;FOLD PLACE 2
;FOLD PROPRIEDADES
Ponto_STR[Pallet_2,Prdt_32BarPacking,2].NumCaixas = 3
Ponto_STR[Pallet_2,Prdt_32BarPacking,2].PickOp = 2
Ponto_STR[Pallet_2,Prdt_32BarPacking,2].ConfGarraOp = 3
Ponto_STR[Pallet_2,Prdt_32BarPacking,2].FechaGarraOp = 0
Ponto_STR[Pallet_2,Prdt_32BarPacking,2].AbreGarraOp = 0
Ponto_STR[Pallet_2,Prdt_32BarPacking,2].SensoresCaixa = 12345
Ponto_STR[Pallet_2,Prdt_32BarPacking,2].TravaGarra = False
Ponto_STR[Pallet_2,Prdt_32BarPacking,2].SkipGoHome = False
Ponto_STR[Pallet_2,Prdt_32BarPacking,2].SkipSobeRelativo = False
Ponto_STR[Pallet_2,Prdt_32BarPacking,2].XApp1Place=P2_32BarPacking_2_App1
Ponto_STR[Pallet_2,Prdt_32BarPacking,2].XApp2Place=P2_32BarPacking_2_App2
Ponto_STR[Pallet_2,Prdt_32BarPacking,2].XPlace=P2_32BarPacking_2_Place
;ENDFOLD
;FOLD OffsetPlace
Ponto_STR[Pallet_2,Prdt_32BarPacking,2].OffsetPlace.X=0
Ponto_STR[Pallet_2,Prdt_32BarPacking,2].OffsetPlace.Y=0
Ponto_STR[Pallet_2,Prdt_32BarPacking,2].OffsetPlace.Z=0
Ponto_STR[Pallet_2,Prdt_32BarPacking,2].OffsetPlace.A=0
Ponto_STR[Pallet_2,Prdt_32BarPacking,2].OffsetPlace.B=0
Ponto_STR[Pallet_2,Prdt_32BarPacking,2].OffsetPlace.C=0
;ENDFOLD
;ENDFOLD

;FOLD PLACE 3
;FOLD PROPRIEDADES
Ponto_STR[Pallet_2,Prdt_32BarPacking,3].NumCaixas = 3
Ponto_STR[Pallet_2,Prdt_32BarPacking,3].PickOp = 2
Ponto_STR[Pallet_2,Prdt_32BarPacking,3].ConfGarraOp = 3
Ponto_STR[Pallet_2,Prdt_32BarPacking,3].FechaGarraOp = 0
Ponto_STR[Pallet_2,Prdt_32BarPacking,3].AbreGarraOp = 0
Ponto_STR[Pallet_2,Prdt_32BarPacking,3].SensoresCaixa = 12345
Ponto_STR[Pallet_2,Prdt_32BarPacking,3].TravaGarra = False
Ponto_STR[Pallet_2,Prdt_32BarPacking,3].SkipGoHome = False
Ponto_STR[Pallet_2,Prdt_32BarPacking,3].SkipSobeRelativo = False
Ponto_STR[Pallet_2,Prdt_32BarPacking,3].XApp1Place=P2_32BarPacking_3_App1
Ponto_STR[Pallet_2,Prdt_32BarPacking,3].XApp2Place=P2_32BarPacking_3_App2
Ponto_STR[Pallet_2,Prdt_32BarPacking,3].XPlace=P2_32BarPacking_3_Place
;ENDFOLD
;FOLD OffsetPlace
Ponto_STR[Pallet_2,Prdt_32BarPacking,3].OffsetPlace.X=0
Ponto_STR[Pallet_2,Prdt_32BarPacking,3].OffsetPlace.Y=0
Ponto_STR[Pallet_2,Prdt_32BarPacking,3].OffsetPlace.Z=0
Ponto_STR[Pallet_2,Prdt_32BarPacking,3].OffsetPlace.A=0
Ponto_STR[Pallet_2,Prdt_32BarPacking,3].OffsetPlace.B=0
Ponto_STR[Pallet_2,Prdt_32BarPacking,3].OffsetPlace.C=0
;ENDFOLD
;ENDFOLD

;ENDFOLD
;ENDFOLD

;FOLD Pallet 2 - Produto 33BarPacking
;FOLD LAYER 1: PLACE 1 ate 2
;FOLD PLACE 1
;FOLD PROPRIEDADES
Ponto_STR[Pallet_2,Prdt_33BarPacking,1].NumCaixas = 3
Ponto_STR[Pallet_2,Prdt_33BarPacking,1].PickOp = 2
Ponto_STR[Pallet_2,Prdt_33BarPacking,1].ConfGarraOp = 2
Ponto_STR[Pallet_2,Prdt_33BarPacking,1].FechaGarraOp = 0
Ponto_STR[Pallet_2,Prdt_33BarPacking,1].AbreGarraOp = 0
Ponto_STR[Pallet_2,Prdt_33BarPacking,1].SensoresCaixa = 12345
Ponto_STR[Pallet_2,Prdt_33BarPacking,1].TravaGarra = False
Ponto_STR[Pallet_2,Prdt_33BarPacking,1].SkipGoHome = False
Ponto_STR[Pallet_2,Prdt_33BarPacking,1].SkipSobeRelativo = False
Ponto_STR[Pallet_2,Prdt_33BarPacking,1].XApp1Place=P2_33BarPacking_1_App1
Ponto_STR[Pallet_2,Prdt_33BarPacking,1].XApp2Place=P2_33BarPacking_1_App2
Ponto_STR[Pallet_2,Prdt_33BarPacking,1].XPlace=P2_33BarPacking_1_Place
;ENDFOLD
;FOLD OffsetPlace
Ponto_STR[Pallet_2,Prdt_33BarPacking,1].OffsetPlace.X=0
Ponto_STR[Pallet_2,Prdt_33BarPacking,1].OffsetPlace.Y=0
Ponto_STR[Pallet_2,Prdt_33BarPacking,1].OffsetPlace.Z=0
Ponto_STR[Pallet_2,Prdt_33BarPacking,1].OffsetPlace.A=0
Ponto_STR[Pallet_2,Prdt_33BarPacking,1].OffsetPlace.B=0
Ponto_STR[Pallet_2,Prdt_33BarPacking,1].OffsetPlace.C=0
;ENDFOLD
;ENDFOLD

;FOLD PLACE 2
;FOLD PROPRIEDADES
Ponto_STR[Pallet_2,Prdt_33BarPacking,2].NumCaixas = 3
Ponto_STR[Pallet_2,Prdt_33BarPacking,2].PickOp = 2
Ponto_STR[Pallet_2,Prdt_33BarPacking,2].ConfGarraOp = 2
Ponto_STR[Pallet_2,Prdt_33BarPacking,2].FechaGarraOp = 0
Ponto_STR[Pallet_2,Prdt_33BarPacking,2].AbreGarraOp = 0
Ponto_STR[Pallet_2,Prdt_33BarPacking,2].SensoresCaixa = 12345
Ponto_STR[Pallet_2,Prdt_33BarPacking,2].TravaGarra = False
Ponto_STR[Pallet_2,Prdt_33BarPacking,2].SkipGoHome = False
Ponto_STR[Pallet_2,Prdt_33BarPacking,2].SkipSobeRelativo = False
Ponto_STR[Pallet_2,Prdt_33BarPacking,2].XApp1Place=P2_33BarPacking_2_App1
Ponto_STR[Pallet_2,Prdt_33BarPacking,2].XApp2Place=P2_33BarPacking_2_App2
Ponto_STR[Pallet_2,Prdt_33BarPacking,2].XPlace=P2_33BarPacking_2_Place
;ENDFOLD
;FOLD OffsetPlace
Ponto_STR[Pallet_2,Prdt_33BarPacking,2].OffsetPlace.X=0
Ponto_STR[Pallet_2,Prdt_33BarPacking,2].OffsetPlace.Y=0
Ponto_STR[Pallet_2,Prdt_33BarPacking,2].OffsetPlace.Z=0
Ponto_STR[Pallet_2,Prdt_33BarPacking,2].OffsetPlace.A=0
Ponto_STR[Pallet_2,Prdt_33BarPacking,2].OffsetPlace.B=0
Ponto_STR[Pallet_2,Prdt_33BarPacking,2].OffsetPlace.C=0
;ENDFOLD
;ENDFOLD

;ENDFOLD
;ENDFOLD

;FOLD Pallet 2 - Produto 34BarPacking
;FOLD LAYER 1: PLACE 1 ate 2
;FOLD PLACE 1
;FOLD PROPRIEDADES
Ponto_STR[Pallet_2,Prdt_34BarPacking,1].NumCaixas = 1
Ponto_STR[Pallet_2,Prdt_34BarPacking,1].PickOp = 3
Ponto_STR[Pallet_2,Prdt_34BarPacking,1].ConfGarraOp = 3
Ponto_STR[Pallet_2,Prdt_34BarPacking,1].FechaGarraOp = 0
Ponto_STR[Pallet_2,Prdt_34BarPacking,1].AbreGarraOp = 0
Ponto_STR[Pallet_2,Prdt_34BarPacking,1].SensoresCaixa = 123
Ponto_STR[Pallet_2,Prdt_34BarPacking,1].TravaGarra = False
Ponto_STR[Pallet_2,Prdt_34BarPacking,1].SkipGoHome = False
Ponto_STR[Pallet_2,Prdt_34BarPacking,1].SkipSobeRelativo = False
Ponto_STR[Pallet_2,Prdt_34BarPacking,1].XApp1Place=P2_34BarPacking_1_App1
Ponto_STR[Pallet_2,Prdt_34BarPacking,1].XApp2Place=P2_34BarPacking_1_App2
Ponto_STR[Pallet_2,Prdt_34BarPacking,1].XPlace=P2_34BarPacking_1_Place
;ENDFOLD
;FOLD OffsetPlace
Ponto_STR[Pallet_2,Prdt_34BarPacking,1].OffsetPlace.X=0
Ponto_STR[Pallet_2,Prdt_34BarPacking,1].OffsetPlace.Y=0
Ponto_STR[Pallet_2,Prdt_34BarPacking,1].OffsetPlace.Z=0
Ponto_STR[Pallet_2,Prdt_34BarPacking,1].OffsetPlace.A=0
Ponto_STR[Pallet_2,Prdt_34BarPacking,1].OffsetPlace.B=0
Ponto_STR[Pallet_2,Prdt_34BarPacking,1].OffsetPlace.C=0
;ENDFOLD
;ENDFOLD

;FOLD PLACE 2
;FOLD PROPRIEDADES
Ponto_STR[Pallet_2,Prdt_34BarPacking,2].NumCaixas = 1
Ponto_STR[Pallet_2,Prdt_34BarPacking,2].PickOp = 3
Ponto_STR[Pallet_2,Prdt_34BarPacking,2].ConfGarraOp = 3
Ponto_STR[Pallet_2,Prdt_34BarPacking,2].FechaGarraOp = 0
Ponto_STR[Pallet_2,Prdt_34BarPacking,2].AbreGarraOp = 0
Ponto_STR[Pallet_2,Prdt_34BarPacking,2].SensoresCaixa = 123
Ponto_STR[Pallet_2,Prdt_34BarPacking,2].TravaGarra = False
Ponto_STR[Pallet_2,Prdt_34BarPacking,2].SkipGoHome = False
Ponto_STR[Pallet_2,Prdt_34BarPacking,2].SkipSobeRelativo = False
Ponto_STR[Pallet_2,Prdt_34BarPacking,2].XApp1Place=P2_34BarPacking_2_App1
Ponto_STR[Pallet_2,Prdt_34BarPacking,2].XApp2Place=P2_34BarPacking_2_App2
Ponto_STR[Pallet_2,Prdt_34BarPacking,2].XPlace=P2_34BarPacking_2_Place
;ENDFOLD
;FOLD OffsetPlace
Ponto_STR[Pallet_2,Prdt_34BarPacking,2].OffsetPlace.X=0
Ponto_STR[Pallet_2,Prdt_34BarPacking,2].OffsetPlace.Y=0
Ponto_STR[Pallet_2,Prdt_34BarPacking,2].OffsetPlace.Z=0
Ponto_STR[Pallet_2,Prdt_34BarPacking,2].OffsetPlace.A=0
Ponto_STR[Pallet_2,Prdt_34BarPacking,2].OffsetPlace.B=0
Ponto_STR[Pallet_2,Prdt_34BarPacking,2].OffsetPlace.C=0
;ENDFOLD
;ENDFOLD

;ENDFOLD
;ENDFOLD

;FOLD Pallet 2 - Produto 9Aero
;FOLD LAYER 1: PLACE 1 ate 2
;FOLD PLACE 1
;FOLD PROPRIEDADES
Ponto_STR[Pallet_2,Prdt_9Aero,1].NumCaixas = 4
Ponto_STR[Pallet_2,Prdt_9Aero,1].PickOp = 3
Ponto_STR[Pallet_2,Prdt_9Aero,1].ConfGarraOp = 3
Ponto_STR[Pallet_2,Prdt_9Aero,1].FechaGarraOp = 0
Ponto_STR[Pallet_2,Prdt_9Aero,1].AbreGarraOp = 0
Ponto_STR[Pallet_2,Prdt_9Aero,1].SensoresCaixa = 123456
Ponto_STR[Pallet_2,Prdt_9Aero,1].TravaGarra = False
Ponto_STR[Pallet_2,Prdt_9Aero,1].SkipGoHome = False
Ponto_STR[Pallet_2,Prdt_9Aero,1].SkipSobeRelativo = False
Ponto_STR[Pallet_2,Prdt_9Aero,1].XApp1Place=P2_9Aero_1_App1
Ponto_STR[Pallet_2,Prdt_9Aero,1].XApp2Place=P2_9Aero_1_App2
Ponto_STR[Pallet_2,Prdt_9Aero,1].XPlace=P2_9Aero_1_Place
;ENDFOLD
;FOLD OffsetPlace
Ponto_STR[Pallet_2,Prdt_9Aero,1].OffsetPlace.X=0
Ponto_STR[Pallet_2,Prdt_9Aero,1].OffsetPlace.Y=0
Ponto_STR[Pallet_2,Prdt_9Aero,1].OffsetPlace.Z=0
Ponto_STR[Pallet_2,Prdt_9Aero,1].OffsetPlace.A=0
Ponto_STR[Pallet_2,Prdt_9Aero,1].OffsetPlace.B=0
Ponto_STR[Pallet_2,Prdt_9Aero,1].OffsetPlace.C=0
;ENDFOLD
;ENDFOLD

;FOLD PLACE 2
;FOLD PROPRIEDADES
Ponto_STR[Pallet_2,Prdt_9Aero,2].NumCaixas = 4
Ponto_STR[Pallet_2,Prdt_9Aero,2].PickOp = 3
Ponto_STR[Pallet_2,Prdt_9Aero,2].ConfGarraOp = 3
Ponto_STR[Pallet_2,Prdt_9Aero,2].FechaGarraOp = 0
Ponto_STR[Pallet_2,Prdt_9Aero,2].AbreGarraOp = 0
Ponto_STR[Pallet_2,Prdt_9Aero,2].SensoresCaixa = 123456
Ponto_STR[Pallet_2,Prdt_9Aero,2].TravaGarra = False
Ponto_STR[Pallet_2,Prdt_9Aero,2].SkipGoHome = False
Ponto_STR[Pallet_2,Prdt_9Aero,2].SkipSobeRelativo = False
Ponto_STR[Pallet_2,Prdt_9Aero,2].XApp1Place=P2_9Aero_2_App1
Ponto_STR[Pallet_2,Prdt_9Aero,2].XApp2Place=P2_9Aero_2_App2
Ponto_STR[Pallet_2,Prdt_9Aero,2].XPlace=P2_9Aero_2_Place
;ENDFOLD
;FOLD OffsetPlace
Ponto_STR[Pallet_2,Prdt_9Aero,2].OffsetPlace.X=0
Ponto_STR[Pallet_2,Prdt_9Aero,2].OffsetPlace.Y=0
Ponto_STR[Pallet_2,Prdt_9Aero,2].OffsetPlace.Z=0
Ponto_STR[Pallet_2,Prdt_9Aero,2].OffsetPlace.A=0
Ponto_STR[Pallet_2,Prdt_9Aero,2].OffsetPlace.B=0
Ponto_STR[Pallet_2,Prdt_9Aero,2].OffsetPlace.C=0
;ENDFOLD
;ENDFOLD

;ENDFOLD
;ENDFOLD

;FOLD Pallet 2 - Produto 23Smarties
;FOLD LAYER 1: PLACE 1 ate 4
;FOLD PLACE 1
;FOLD PROPRIEDADES
Ponto_STR[Pallet_2,Prdt_23Smarties,1].NumCaixas = 2
Ponto_STR[Pallet_2,Prdt_23Smarties,1].PickOp = 4
Ponto_STR[Pallet_2,Prdt_23Smarties,1].ConfGarraOp = 4
Ponto_STR[Pallet_2,Prdt_23Smarties,1].FechaGarraOp = 0
Ponto_STR[Pallet_2,Prdt_23Smarties,1].AbreGarraOp = 0
Ponto_STR[Pallet_2,Prdt_23Smarties,1].SensoresCaixa = 456
Ponto_STR[Pallet_2,Prdt_23Smarties,1].TravaGarra = False
Ponto_STR[Pallet_2,Prdt_23Smarties,1].SkipGoHome = False
Ponto_STR[Pallet_2,Prdt_23Smarties,1].SkipSobeRelativo = False
Ponto_STR[Pallet_2,Prdt_23Smarties,1].XApp1Place=P2_23Smarties_1_App1
Ponto_STR[Pallet_2,Prdt_23Smarties,1].XApp2Place=P2_23Smarties_1_App2
Ponto_STR[Pallet_2,Prdt_23Smarties,1].XPlace=P2_23Smarties_1_Place
;ENDFOLD
;FOLD OffsetPlace
Ponto_STR[Pallet_2,Prdt_23Smarties,1].OffsetPlace.X=0
Ponto_STR[Pallet_2,Prdt_23Smarties,1].OffsetPlace.Y=0
Ponto_STR[Pallet_2,Prdt_23Smarties,1].OffsetPlace.Z=0
Ponto_STR[Pallet_2,Prdt_23Smarties,1].OffsetPlace.A=0
Ponto_STR[Pallet_2,Prdt_23Smarties,1].OffsetPlace.B=0
Ponto_STR[Pallet_2,Prdt_23Smarties,1].OffsetPlace.C=0
;ENDFOLD
;ENDFOLD

;FOLD PLACE 2
;FOLD PROPRIEDADES
Ponto_STR[Pallet_2,Prdt_23Smarties,2].NumCaixas = 3
Ponto_STR[Pallet_2,Prdt_23Smarties,2].PickOp = 4
Ponto_STR[Pallet_2,Prdt_23Smarties,2].ConfGarraOp = 4
Ponto_STR[Pallet_2,Prdt_23Smarties,2].FechaGarraOp = 0
Ponto_STR[Pallet_2,Prdt_23Smarties,2].AbreGarraOp = 0
Ponto_STR[Pallet_2,Prdt_23Smarties,2].SensoresCaixa = 3456
Ponto_STR[Pallet_2,Prdt_23Smarties,2].TravaGarra = False
Ponto_STR[Pallet_2,Prdt_23Smarties,2].SkipGoHome = False
Ponto_STR[Pallet_2,Prdt_23Smarties,2].SkipSobeRelativo = False
Ponto_STR[Pallet_2,Prdt_23Smarties,2].XApp1Place=P2_23Smarties_2_App1
Ponto_STR[Pallet_2,Prdt_23Smarties,2].XApp2Place=P2_23Smarties_2_App2
Ponto_STR[Pallet_2,Prdt_23Smarties,2].XPlace=P2_23Smarties_2_Place
;ENDFOLD
;FOLD OffsetPlace
Ponto_STR[Pallet_2,Prdt_23Smarties,2].OffsetPlace.X=0
Ponto_STR[Pallet_2,Prdt_23Smarties,2].OffsetPlace.Y=0
Ponto_STR[Pallet_2,Prdt_23Smarties,2].OffsetPlace.Z=0
Ponto_STR[Pallet_2,Prdt_23Smarties,2].OffsetPlace.A=0
Ponto_STR[Pallet_2,Prdt_23Smarties,2].OffsetPlace.B=0
Ponto_STR[Pallet_2,Prdt_23Smarties,2].OffsetPlace.C=0
;ENDFOLD
;ENDFOLD

;FOLD PLACE 3
;FOLD PROPRIEDADES
Ponto_STR[Pallet_2,Prdt_23Smarties,3].NumCaixas = 2
Ponto_STR[Pallet_2,Prdt_23Smarties,3].PickOp = 4
Ponto_STR[Pallet_2,Prdt_23Smarties,3].ConfGarraOp = 4
Ponto_STR[Pallet_2,Prdt_23Smarties,3].FechaGarraOp = 0
Ponto_STR[Pallet_2,Prdt_23Smarties,3].AbreGarraOp = 0
Ponto_STR[Pallet_2,Prdt_23Smarties,3].SensoresCaixa = 456
Ponto_STR[Pallet_2,Prdt_23Smarties,3].TravaGarra = False
Ponto_STR[Pallet_2,Prdt_23Smarties,3].SkipGoHome = False
Ponto_STR[Pallet_2,Prdt_23Smarties,3].SkipSobeRelativo = False
Ponto_STR[Pallet_2,Prdt_23Smarties,3].XApp1Place=P2_23Smarties_3_App1
Ponto_STR[Pallet_2,Prdt_23Smarties,3].XApp2Place=P2_23Smarties_3_App2
Ponto_STR[Pallet_2,Prdt_23Smarties,3].XPlace=P2_23Smarties_3_Place
;ENDFOLD
;FOLD OffsetPlace
Ponto_STR[Pallet_2,Prdt_23Smarties,3].OffsetPlace.X=0
Ponto_STR[Pallet_2,Prdt_23Smarties,3].OffsetPlace.Y=0
Ponto_STR[Pallet_2,Prdt_23Smarties,3].OffsetPlace.Z=0
Ponto_STR[Pallet_2,Prdt_23Smarties,3].OffsetPlace.A=0
Ponto_STR[Pallet_2,Prdt_23Smarties,3].OffsetPlace.B=0
Ponto_STR[Pallet_2,Prdt_23Smarties,3].OffsetPlace.C=0
;ENDFOLD
;ENDFOLD

;FOLD PLACE 4
;FOLD PROPRIEDADES
Ponto_STR[Pallet_2,Prdt_23Smarties,4].NumCaixas = 3
Ponto_STR[Pallet_2,Prdt_23Smarties,4].PickOp = 4
Ponto_STR[Pallet_2,Prdt_23Smarties,4].ConfGarraOp = 4
Ponto_STR[Pallet_2,Prdt_23Smarties,4].FechaGarraOp = 0
Ponto_STR[Pallet_2,Prdt_23Smarties,4].AbreGarraOp = 0
Ponto_STR[Pallet_2,Prdt_23Smarties,4].SensoresCaixa = 3456
Ponto_STR[Pallet_2,Prdt_23Smarties,4].TravaGarra = False
Ponto_STR[Pallet_2,Prdt_23Smarties,4].SkipGoHome = False
Ponto_STR[Pallet_2,Prdt_23Smarties,4].SkipSobeRelativo = False
Ponto_STR[Pallet_2,Prdt_23Smarties,4].XApp1Place=P2_23Smarties_4_App1
Ponto_STR[Pallet_2,Prdt_23Smarties,4].XApp2Place=P2_23Smarties_4_App2
Ponto_STR[Pallet_2,Prdt_23Smarties,4].XPlace=P2_23Smarties_4_Place
;ENDFOLD
;FOLD OffsetPlace
Ponto_STR[Pallet_2,Prdt_23Smarties,4].OffsetPlace.X=0
Ponto_STR[Pallet_2,Prdt_23Smarties,4].OffsetPlace.Y=0
Ponto_STR[Pallet_2,Prdt_23Smarties,4].OffsetPlace.Z=0
Ponto_STR[Pallet_2,Prdt_23Smarties,4].OffsetPlace.A=0
Ponto_STR[Pallet_2,Prdt_23Smarties,4].OffsetPlace.B=0
Ponto_STR[Pallet_2,Prdt_23Smarties,4].OffsetPlace.C=0
;ENDFOLD
;ENDFOLD

;ENDFOLD
;FOLD LAYER 2: PLACE 5 ate 8
;FOLD PLACE 5
;FOLD PROPRIEDADES
Ponto_STR[Pallet_2,Prdt_23Smarties,5].NumCaixas = 2
Ponto_STR[Pallet_2,Prdt_23Smarties,5].PickOp = 5
Ponto_STR[Pallet_2,Prdt_23Smarties,5].ConfGarraOp = 4
Ponto_STR[Pallet_2,Prdt_23Smarties,5].FechaGarraOp = 0
Ponto_STR[Pallet_2,Prdt_23Smarties,5].AbreGarraOp = 0
Ponto_STR[Pallet_2,Prdt_23Smarties,5].SensoresCaixa = 123
Ponto_STR[Pallet_2,Prdt_23Smarties,5].TravaGarra = False
Ponto_STR[Pallet_2,Prdt_23Smarties,5].SkipGoHome = False
Ponto_STR[Pallet_2,Prdt_23Smarties,5].SkipSobeRelativo = False
Ponto_STR[Pallet_2,Prdt_23Smarties,5].XApp1Place=P2_23Smarties_5_App1
Ponto_STR[Pallet_2,Prdt_23Smarties,5].XApp2Place=P2_23Smarties_5_App2
Ponto_STR[Pallet_2,Prdt_23Smarties,5].XPlace=P2_23Smarties_5_Place
;ENDFOLD
;FOLD OffsetPlace
Ponto_STR[Pallet_2,Prdt_23Smarties,5].OffsetPlace.X=0
Ponto_STR[Pallet_2,Prdt_23Smarties,5].OffsetPlace.Y=0
Ponto_STR[Pallet_2,Prdt_23Smarties,5].OffsetPlace.Z=0
Ponto_STR[Pallet_2,Prdt_23Smarties,5].OffsetPlace.A=0
Ponto_STR[Pallet_2,Prdt_23Smarties,5].OffsetPlace.B=0
Ponto_STR[Pallet_2,Prdt_23Smarties,5].OffsetPlace.C=0
;ENDFOLD
;ENDFOLD

;FOLD PLACE 6
;FOLD PROPRIEDADES
Ponto_STR[Pallet_2,Prdt_23Smarties,6].NumCaixas = 3
Ponto_STR[Pallet_2,Prdt_23Smarties,6].PickOp = 5
Ponto_STR[Pallet_2,Prdt_23Smarties,6].ConfGarraOp = 4
Ponto_STR[Pallet_2,Prdt_23Smarties,6].FechaGarraOp = 0
Ponto_STR[Pallet_2,Prdt_23Smarties,6].AbreGarraOp = 0
Ponto_STR[Pallet_2,Prdt_23Smarties,6].SensoresCaixa = 1234
Ponto_STR[Pallet_2,Prdt_23Smarties,6].TravaGarra = False
Ponto_STR[Pallet_2,Prdt_23Smarties,6].SkipGoHome = False
Ponto_STR[Pallet_2,Prdt_23Smarties,6].SkipSobeRelativo = False
Ponto_STR[Pallet_2,Prdt_23Smarties,6].XApp1Place=P2_23Smarties_6_App1
Ponto_STR[Pallet_2,Prdt_23Smarties,6].XApp2Place=P2_23Smarties_6_App2
Ponto_STR[Pallet_2,Prdt_23Smarties,6].XPlace=P2_23Smarties_6_Place
;ENDFOLD
;FOLD OffsetPlace
Ponto_STR[Pallet_2,Prdt_23Smarties,6].OffsetPlace.X=0
Ponto_STR[Pallet_2,Prdt_23Smarties,6].OffsetPlace.Y=0
Ponto_STR[Pallet_2,Prdt_23Smarties,6].OffsetPlace.Z=0
Ponto_STR[Pallet_2,Prdt_23Smarties,6].OffsetPlace.A=0
Ponto_STR[Pallet_2,Prdt_23Smarties,6].OffsetPlace.B=0
Ponto_STR[Pallet_2,Prdt_23Smarties,6].OffsetPlace.C=0
;ENDFOLD
;ENDFOLD

;FOLD PLACE 7
;FOLD PROPRIEDADES
Ponto_STR[Pallet_2,Prdt_23Smarties,7].NumCaixas = 2
Ponto_STR[Pallet_2,Prdt_23Smarties,7].PickOp = 5
Ponto_STR[Pallet_2,Prdt_23Smarties,7].ConfGarraOp = 4
Ponto_STR[Pallet_2,Prdt_23Smarties,7].FechaGarraOp = 0
Ponto_STR[Pallet_2,Prdt_23Smarties,7].AbreGarraOp = 0
Ponto_STR[Pallet_2,Prdt_23Smarties,7].SensoresCaixa = 123
Ponto_STR[Pallet_2,Prdt_23Smarties,7].TravaGarra = False
Ponto_STR[Pallet_2,Prdt_23Smarties,7].SkipGoHome = False
Ponto_STR[Pallet_2,Prdt_23Smarties,7].SkipSobeRelativo = False
Ponto_STR[Pallet_2,Prdt_23Smarties,7].XApp1Place=P2_23Smarties_7_App1
Ponto_STR[Pallet_2,Prdt_23Smarties,7].XApp2Place=P2_23Smarties_7_App2
Ponto_STR[Pallet_2,Prdt_23Smarties,7].XPlace=P2_23Smarties_7_Place
;ENDFOLD
;FOLD OffsetPlace
Ponto_STR[Pallet_2,Prdt_23Smarties,7].OffsetPlace.X=0
Ponto_STR[Pallet_2,Prdt_23Smarties,7].OffsetPlace.Y=0
Ponto_STR[Pallet_2,Prdt_23Smarties,7].OffsetPlace.Z=0
Ponto_STR[Pallet_2,Prdt_23Smarties,7].OffsetPlace.A=0
Ponto_STR[Pallet_2,Prdt_23Smarties,7].OffsetPlace.B=0
Ponto_STR[Pallet_2,Prdt_23Smarties,7].OffsetPlace.C=0
;ENDFOLD
;ENDFOLD

;FOLD PLACE 8
;FOLD PROPRIEDADES
Ponto_STR[Pallet_2,Prdt_23Smarties,8].NumCaixas = 3
Ponto_STR[Pallet_2,Prdt_23Smarties,8].PickOp = 5
Ponto_STR[Pallet_2,Prdt_23Smarties,8].ConfGarraOp = 4
Ponto_STR[Pallet_2,Prdt_23Smarties,8].FechaGarraOp = 0
Ponto_STR[Pallet_2,Prdt_23Smarties,8].AbreGarraOp = 0
Ponto_STR[Pallet_2,Prdt_23Smarties,8].SensoresCaixa = 1234
Ponto_STR[Pallet_2,Prdt_23Smarties,8].TravaGarra = False
Ponto_STR[Pallet_2,Prdt_23Smarties,8].SkipGoHome = False
Ponto_STR[Pallet_2,Prdt_23Smarties,8].SkipSobeRelativo = False
Ponto_STR[Pallet_2,Prdt_23Smarties,8].XApp1Place=P2_23Smarties_8_App1
Ponto_STR[Pallet_2,Prdt_23Smarties,8].XApp2Place=P2_23Smarties_8_App2
Ponto_STR[Pallet_2,Prdt_23Smarties,8].XPlace=P2_23Smarties_8_Place
;ENDFOLD
;FOLD OffsetPlace
Ponto_STR[Pallet_2,Prdt_23Smarties,8].OffsetPlace.X=0
Ponto_STR[Pallet_2,Prdt_23Smarties,8].OffsetPlace.Y=0
Ponto_STR[Pallet_2,Prdt_23Smarties,8].OffsetPlace.Z=0
Ponto_STR[Pallet_2,Prdt_23Smarties,8].OffsetPlace.A=0
Ponto_STR[Pallet_2,Prdt_23Smarties,8].OffsetPlace.B=0
Ponto_STR[Pallet_2,Prdt_23Smarties,8].OffsetPlace.C=0
;ENDFOLD
;ENDFOLD

;ENDFOLD
;ENDFOLD

;FOLD Pallet 2 - Produto 10CoffeCrisp
;FOLD LAYER 1: PLACE 1 ate 4
;FOLD PLACE 1
;FOLD PROPRIEDADES
Ponto_STR[Pallet_2,Prdt_10CoffeCrisp,1].NumCaixas = 1
Ponto_STR[Pallet_2,Prdt_10CoffeCrisp,1].PickOp = 6
Ponto_STR[Pallet_2,Prdt_10CoffeCrisp,1].ConfGarraOp = 0
Ponto_STR[Pallet_2,Prdt_10CoffeCrisp,1].FechaGarraOp = 0
Ponto_STR[Pallet_2,Prdt_10CoffeCrisp,1].AbreGarraOp = 0
Ponto_STR[Pallet_2,Prdt_10CoffeCrisp,1].SensoresCaixa = 56
Ponto_STR[Pallet_2,Prdt_10CoffeCrisp,1].TravaGarra = False
Ponto_STR[Pallet_2,Prdt_10CoffeCrisp,1].SkipGoHome = False
Ponto_STR[Pallet_2,Prdt_10CoffeCrisp,1].SkipSobeRelativo = False
Ponto_STR[Pallet_2,Prdt_10CoffeCrisp,1].XApp1Place=P2_10CoffeCrisp_1_App1
Ponto_STR[Pallet_2,Prdt_10CoffeCrisp,1].XApp2Place=P2_10CoffeCrisp_1_App2
Ponto_STR[Pallet_2,Prdt_10CoffeCrisp,1].XPlace=P2_10CoffeCrisp_1_Place
;ENDFOLD
;FOLD OffsetPlace
Ponto_STR[Pallet_2,Prdt_10CoffeCrisp,1].OffsetPlace.X=0
Ponto_STR[Pallet_2,Prdt_10CoffeCrisp,1].OffsetPlace.Y=0
Ponto_STR[Pallet_2,Prdt_10CoffeCrisp,1].OffsetPlace.Z=0
Ponto_STR[Pallet_2,Prdt_10CoffeCrisp,1].OffsetPlace.A=0
Ponto_STR[Pallet_2,Prdt_10CoffeCrisp,1].OffsetPlace.B=0
Ponto_STR[Pallet_2,Prdt_10CoffeCrisp,1].OffsetPlace.C=0
;ENDFOLD
;ENDFOLD

;FOLD PLACE 2
;FOLD PROPRIEDADES
Ponto_STR[Pallet_2,Prdt_10CoffeCrisp,2].NumCaixas = 1
Ponto_STR[Pallet_2,Prdt_10CoffeCrisp,2].PickOp = 6
Ponto_STR[Pallet_2,Prdt_10CoffeCrisp,2].ConfGarraOp = 0
Ponto_STR[Pallet_2,Prdt_10CoffeCrisp,2].FechaGarraOp = 0
Ponto_STR[Pallet_2,Prdt_10CoffeCrisp,2].AbreGarraOp = 0
Ponto_STR[Pallet_2,Prdt_10CoffeCrisp,2].SensoresCaixa = 56
Ponto_STR[Pallet_2,Prdt_10CoffeCrisp,2].TravaGarra = False
Ponto_STR[Pallet_2,Prdt_10CoffeCrisp,2].SkipGoHome = False
Ponto_STR[Pallet_2,Prdt_10CoffeCrisp,2].SkipSobeRelativo = False
Ponto_STR[Pallet_2,Prdt_10CoffeCrisp,2].XApp1Place=P2_10CoffeCrisp_2_App1
Ponto_STR[Pallet_2,Prdt_10CoffeCrisp,2].XApp2Place=P2_10CoffeCrisp_2_App2
Ponto_STR[Pallet_2,Prdt_10CoffeCrisp,2].XPlace=P2_10CoffeCrisp_2_Place
;ENDFOLD
;FOLD OffsetPlace
Ponto_STR[Pallet_2,Prdt_10CoffeCrisp,2].OffsetPlace.X=0
Ponto_STR[Pallet_2,Prdt_10CoffeCrisp,2].OffsetPlace.Y=0
Ponto_STR[Pallet_2,Prdt_10CoffeCrisp,2].OffsetPlace.Z=0
Ponto_STR[Pallet_2,Prdt_10CoffeCrisp,2].OffsetPlace.A=0
Ponto_STR[Pallet_2,Prdt_10CoffeCrisp,2].OffsetPlace.B=0
Ponto_STR[Pallet_2,Prdt_10CoffeCrisp,2].OffsetPlace.C=0
;ENDFOLD
;ENDFOLD

;FOLD PLACE 3
;FOLD PROPRIEDADES
Ponto_STR[Pallet_2,Prdt_10CoffeCrisp,3].NumCaixas = 3
Ponto_STR[Pallet_2,Prdt_10CoffeCrisp,3].PickOp = 1
Ponto_STR[Pallet_2,Prdt_10CoffeCrisp,3].ConfGarraOp = 0
Ponto_STR[Pallet_2,Prdt_10CoffeCrisp,3].FechaGarraOp = 0
Ponto_STR[Pallet_2,Prdt_10CoffeCrisp,3].AbreGarraOp = 0
Ponto_STR[Pallet_2,Prdt_10CoffeCrisp,3].SensoresCaixa = 12345
Ponto_STR[Pallet_2,Prdt_10CoffeCrisp,3].TravaGarra = False
Ponto_STR[Pallet_2,Prdt_10CoffeCrisp,3].SkipGoHome = False
Ponto_STR[Pallet_2,Prdt_10CoffeCrisp,3].SkipSobeRelativo = False
Ponto_STR[Pallet_2,Prdt_10CoffeCrisp,3].XApp1Place=P2_10CoffeCrisp_3_App1
Ponto_STR[Pallet_2,Prdt_10CoffeCrisp,3].XApp2Place=P2_10CoffeCrisp_3_App2
Ponto_STR[Pallet_2,Prdt_10CoffeCrisp,3].XPlace=P2_10CoffeCrisp_3_Place
;ENDFOLD
;FOLD OffsetPlace
Ponto_STR[Pallet_2,Prdt_10CoffeCrisp,3].OffsetPlace.X=0
Ponto_STR[Pallet_2,Prdt_10CoffeCrisp,3].OffsetPlace.Y=0
Ponto_STR[Pallet_2,Prdt_10CoffeCrisp,3].OffsetPlace.Z=0
Ponto_STR[Pallet_2,Prdt_10CoffeCrisp,3].OffsetPlace.A=0
Ponto_STR[Pallet_2,Prdt_10CoffeCrisp,3].OffsetPlace.B=0
Ponto_STR[Pallet_2,Prdt_10CoffeCrisp,3].OffsetPlace.C=0
;ENDFOLD
;ENDFOLD

;FOLD PLACE 4
;FOLD PROPRIEDADES
Ponto_STR[Pallet_2,Prdt_10CoffeCrisp,4].NumCaixas = 3
Ponto_STR[Pallet_2,Prdt_10CoffeCrisp,4].PickOp = 1
Ponto_STR[Pallet_2,Prdt_10CoffeCrisp,4].ConfGarraOp = 0
Ponto_STR[Pallet_2,Prdt_10CoffeCrisp,4].FechaGarraOp = 0
Ponto_STR[Pallet_2,Prdt_10CoffeCrisp,4].AbreGarraOp = 0
Ponto_STR[Pallet_2,Prdt_10CoffeCrisp,4].SensoresCaixa = 12345
Ponto_STR[Pallet_2,Prdt_10CoffeCrisp,4].TravaGarra = False
Ponto_STR[Pallet_2,Prdt_10CoffeCrisp,4].SkipGoHome = False
Ponto_STR[Pallet_2,Prdt_10CoffeCrisp,4].SkipSobeRelativo = False
Ponto_STR[Pallet_2,Prdt_10CoffeCrisp,4].XApp1Place=P2_10CoffeCrisp_4_App1
Ponto_STR[Pallet_2,Prdt_10CoffeCrisp,4].XApp2Place=P2_10CoffeCrisp_4_App2
Ponto_STR[Pallet_2,Prdt_10CoffeCrisp,4].XPlace=P2_10CoffeCrisp_4_Place
;ENDFOLD
;FOLD OffsetPlace
Ponto_STR[Pallet_2,Prdt_10CoffeCrisp,4].OffsetPlace.X=0
Ponto_STR[Pallet_2,Prdt_10CoffeCrisp,4].OffsetPlace.Y=0
Ponto_STR[Pallet_2,Prdt_10CoffeCrisp,4].OffsetPlace.Z=0
Ponto_STR[Pallet_2,Prdt_10CoffeCrisp,4].OffsetPlace.A=0
Ponto_STR[Pallet_2,Prdt_10CoffeCrisp,4].OffsetPlace.B=0
Ponto_STR[Pallet_2,Prdt_10CoffeCrisp,4].OffsetPlace.C=0
;ENDFOLD
;ENDFOLD

;ENDFOLD
;FOLD LAYER 2: PLACE 5 ate 8
;FOLD PLACE 5
;FOLD PROPRIEDADES
Ponto_STR[Pallet_2,Prdt_10CoffeCrisp,5].NumCaixas = 1
Ponto_STR[Pallet_2,Prdt_10CoffeCrisp,5].PickOp = 3
Ponto_STR[Pallet_2,Prdt_10CoffeCrisp,5].ConfGarraOp = 3
Ponto_STR[Pallet_2,Prdt_10CoffeCrisp,5].FechaGarraOp = 0
Ponto_STR[Pallet_2,Prdt_10CoffeCrisp,5].AbreGarraOp = 0
Ponto_STR[Pallet_2,Prdt_10CoffeCrisp,5].SensoresCaixa = 12
Ponto_STR[Pallet_2,Prdt_10CoffeCrisp,5].TravaGarra = False
Ponto_STR[Pallet_2,Prdt_10CoffeCrisp,5].SkipGoHome = False
Ponto_STR[Pallet_2,Prdt_10CoffeCrisp,5].SkipSobeRelativo = False
Ponto_STR[Pallet_2,Prdt_10CoffeCrisp,5].XApp1Place=P2_10CoffeCrisp_5_App1
Ponto_STR[Pallet_2,Prdt_10CoffeCrisp,5].XApp2Place=P2_10CoffeCrisp_5_App2
Ponto_STR[Pallet_2,Prdt_10CoffeCrisp,5].XPlace=P2_10CoffeCrisp_5_Place
;ENDFOLD
;FOLD OffsetPlace
Ponto_STR[Pallet_2,Prdt_10CoffeCrisp,5].OffsetPlace.X=0
Ponto_STR[Pallet_2,Prdt_10CoffeCrisp,5].OffsetPlace.Y=0
Ponto_STR[Pallet_2,Prdt_10CoffeCrisp,5].OffsetPlace.Z=0
Ponto_STR[Pallet_2,Prdt_10CoffeCrisp,5].OffsetPlace.A=0
Ponto_STR[Pallet_2,Prdt_10CoffeCrisp,5].OffsetPlace.B=0
Ponto_STR[Pallet_2,Prdt_10CoffeCrisp,5].OffsetPlace.C=0
;ENDFOLD
;ENDFOLD

;FOLD PLACE 6
;FOLD PROPRIEDADES
Ponto_STR[Pallet_2,Prdt_10CoffeCrisp,6].NumCaixas = 1
Ponto_STR[Pallet_2,Prdt_10CoffeCrisp,6].PickOp = 3
Ponto_STR[Pallet_2,Prdt_10CoffeCrisp,6].ConfGarraOp = 3
Ponto_STR[Pallet_2,Prdt_10CoffeCrisp,6].FechaGarraOp = 0
Ponto_STR[Pallet_2,Prdt_10CoffeCrisp,6].AbreGarraOp = 0
Ponto_STR[Pallet_2,Prdt_10CoffeCrisp,6].SensoresCaixa = 12
Ponto_STR[Pallet_2,Prdt_10CoffeCrisp,6].TravaGarra = False
Ponto_STR[Pallet_2,Prdt_10CoffeCrisp,6].SkipGoHome = False
Ponto_STR[Pallet_2,Prdt_10CoffeCrisp,6].SkipSobeRelativo = False
Ponto_STR[Pallet_2,Prdt_10CoffeCrisp,6].XApp1Place=P2_10CoffeCrisp_6_App1
Ponto_STR[Pallet_2,Prdt_10CoffeCrisp,6].XApp2Place=P2_10CoffeCrisp_6_App2
Ponto_STR[Pallet_2,Prdt_10CoffeCrisp,6].XPlace=P2_10CoffeCrisp_6_Place
;ENDFOLD
;FOLD OffsetPlace
Ponto_STR[Pallet_2,Prdt_10CoffeCrisp,6].OffsetPlace.X=0
Ponto_STR[Pallet_2,Prdt_10CoffeCrisp,6].OffsetPlace.Y=0
Ponto_STR[Pallet_2,Prdt_10CoffeCrisp,6].OffsetPlace.Z=0
Ponto_STR[Pallet_2,Prdt_10CoffeCrisp,6].OffsetPlace.A=0
Ponto_STR[Pallet_2,Prdt_10CoffeCrisp,6].OffsetPlace.B=0
Ponto_STR[Pallet_2,Prdt_10CoffeCrisp,6].OffsetPlace.C=0
;ENDFOLD
;ENDFOLD

;FOLD PLACE 7
;FOLD PROPRIEDADES
Ponto_STR[Pallet_2,Prdt_10CoffeCrisp,7].NumCaixas = 3
Ponto_STR[Pallet_2,Prdt_10CoffeCrisp,7].PickOp = 1
Ponto_STR[Pallet_2,Prdt_10CoffeCrisp,7].ConfGarraOp = 0
Ponto_STR[Pallet_2,Prdt_10CoffeCrisp,7].FechaGarraOp = 0
Ponto_STR[Pallet_2,Prdt_10CoffeCrisp,7].AbreGarraOp = 1
Ponto_STR[Pallet_2,Prdt_10CoffeCrisp,7].SensoresCaixa = 12345
Ponto_STR[Pallet_2,Prdt_10CoffeCrisp,7].TravaGarra = True
Ponto_STR[Pallet_2,Prdt_10CoffeCrisp,7].SkipGoHome = False
Ponto_STR[Pallet_2,Prdt_10CoffeCrisp,7].SkipSobeRelativo = False
Ponto_STR[Pallet_2,Prdt_10CoffeCrisp,7].XApp1Place=P2_10CoffeCrisp_7_App1
Ponto_STR[Pallet_2,Prdt_10CoffeCrisp,7].XApp2Place=P2_10CoffeCrisp_7_App2
Ponto_STR[Pallet_2,Prdt_10CoffeCrisp,7].XPlace=P2_10CoffeCrisp_7_Place
;ENDFOLD
;FOLD OffsetPlace
Ponto_STR[Pallet_2,Prdt_10CoffeCrisp,7].OffsetPlace.X=0
Ponto_STR[Pallet_2,Prdt_10CoffeCrisp,7].OffsetPlace.Y=0
Ponto_STR[Pallet_2,Prdt_10CoffeCrisp,7].OffsetPlace.Z=0
Ponto_STR[Pallet_2,Prdt_10CoffeCrisp,7].OffsetPlace.A=0
Ponto_STR[Pallet_2,Prdt_10CoffeCrisp,7].OffsetPlace.B=0
Ponto_STR[Pallet_2,Prdt_10CoffeCrisp,7].OffsetPlace.C=0
;ENDFOLD
;ENDFOLD

;FOLD PLACE 8
;FOLD PROPRIEDADES
Ponto_STR[Pallet_2,Prdt_10CoffeCrisp,8].NumCaixas = 3
Ponto_STR[Pallet_2,Prdt_10CoffeCrisp,8].PickOp = 1
Ponto_STR[Pallet_2,Prdt_10CoffeCrisp,8].ConfGarraOp = 0
Ponto_STR[Pallet_2,Prdt_10CoffeCrisp,8].FechaGarraOp = 0
Ponto_STR[Pallet_2,Prdt_10CoffeCrisp,8].AbreGarraOp = 1
Ponto_STR[Pallet_2,Prdt_10CoffeCrisp,8].SensoresCaixa = 12345
Ponto_STR[Pallet_2,Prdt_10CoffeCrisp,8].TravaGarra = True
Ponto_STR[Pallet_2,Prdt_10CoffeCrisp,8].SkipGoHome = False
Ponto_STR[Pallet_2,Prdt_10CoffeCrisp,8].SkipSobeRelativo = False
Ponto_STR[Pallet_2,Prdt_10CoffeCrisp,8].XApp1Place=P2_10CoffeCrisp_8_App1
Ponto_STR[Pallet_2,Prdt_10CoffeCrisp,8].XApp2Place=P2_10CoffeCrisp_8_App2
Ponto_STR[Pallet_2,Prdt_10CoffeCrisp,8].XPlace=P2_10CoffeCrisp_8_Place
;ENDFOLD
;FOLD OffsetPlace
Ponto_STR[Pallet_2,Prdt_10CoffeCrisp,8].OffsetPlace.X=0
Ponto_STR[Pallet_2,Prdt_10CoffeCrisp,8].OffsetPlace.Y=0
Ponto_STR[Pallet_2,Prdt_10CoffeCrisp,8].OffsetPlace.Z=0
Ponto_STR[Pallet_2,Prdt_10CoffeCrisp,8].OffsetPlace.A=0
Ponto_STR[Pallet_2,Prdt_10CoffeCrisp,8].OffsetPlace.B=0
Ponto_STR[Pallet_2,Prdt_10CoffeCrisp,8].OffsetPlace.C=0
;ENDFOLD
;ENDFOLD

;ENDFOLD
;ENDFOLD

;FOLD Pallet 2 - Produto 19KitKat
;FOLD LAYER 1: PLACE 1 ate 6
;FOLD PLACE 1
;FOLD PROPRIEDADES
Ponto_STR[Pallet_2,Prdt_19KitKat,1].NumCaixas = 1
Ponto_STR[Pallet_2,Prdt_19KitKat,1].PickOp = 6
Ponto_STR[Pallet_2,Prdt_19KitKat,1].ConfGarraOp = 0
Ponto_STR[Pallet_2,Prdt_19KitKat,1].FechaGarraOp = 0
Ponto_STR[Pallet_2,Prdt_19KitKat,1].AbreGarraOp = 0
Ponto_STR[Pallet_2,Prdt_19KitKat,1].SensoresCaixa = 6
Ponto_STR[Pallet_2,Prdt_19KitKat,1].TravaGarra = False
Ponto_STR[Pallet_2,Prdt_19KitKat,1].SkipGoHome = False
Ponto_STR[Pallet_2,Prdt_19KitKat,1].SkipSobeRelativo = False
Ponto_STR[Pallet_2,Prdt_19KitKat,1].XApp1Place=P2_19KitKat_1_App1
Ponto_STR[Pallet_2,Prdt_19KitKat,1].XApp2Place=P2_19KitKat_1_App2
Ponto_STR[Pallet_2,Prdt_19KitKat,1].XPlace=P2_19KitKat_1_Place
;ENDFOLD
;FOLD OffsetPlace
Ponto_STR[Pallet_2,Prdt_19KitKat,1].OffsetPlace.X=0
Ponto_STR[Pallet_2,Prdt_19KitKat,1].OffsetPlace.Y=0
Ponto_STR[Pallet_2,Prdt_19KitKat,1].OffsetPlace.Z=0
Ponto_STR[Pallet_2,Prdt_19KitKat,1].OffsetPlace.A=0
Ponto_STR[Pallet_2,Prdt_19KitKat,1].OffsetPlace.B=0
Ponto_STR[Pallet_2,Prdt_19KitKat,1].OffsetPlace.C=0
;ENDFOLD
;ENDFOLD

;FOLD PLACE 2
;FOLD PROPRIEDADES
Ponto_STR[Pallet_2,Prdt_19KitKat,2].NumCaixas = 1
Ponto_STR[Pallet_2,Prdt_19KitKat,2].PickOp = 6
Ponto_STR[Pallet_2,Prdt_19KitKat,2].ConfGarraOp = 0
Ponto_STR[Pallet_2,Prdt_19KitKat,2].FechaGarraOp = 0
Ponto_STR[Pallet_2,Prdt_19KitKat,2].AbreGarraOp = 0
Ponto_STR[Pallet_2,Prdt_19KitKat,2].SensoresCaixa = 6
Ponto_STR[Pallet_2,Prdt_19KitKat,2].TravaGarra = False
Ponto_STR[Pallet_2,Prdt_19KitKat,2].SkipGoHome = False
Ponto_STR[Pallet_2,Prdt_19KitKat,2].SkipSobeRelativo = False
Ponto_STR[Pallet_2,Prdt_19KitKat,2].XApp1Place=P2_19KitKat_2_App1
Ponto_STR[Pallet_2,Prdt_19KitKat,2].XApp2Place=P2_19KitKat_2_App2
Ponto_STR[Pallet_2,Prdt_19KitKat,2].XPlace=P2_19KitKat_2_Place
;ENDFOLD
;FOLD OffsetPlace
Ponto_STR[Pallet_2,Prdt_19KitKat,2].OffsetPlace.X=0
Ponto_STR[Pallet_2,Prdt_19KitKat,2].OffsetPlace.Y=0
Ponto_STR[Pallet_2,Prdt_19KitKat,2].OffsetPlace.Z=0
Ponto_STR[Pallet_2,Prdt_19KitKat,2].OffsetPlace.A=0
Ponto_STR[Pallet_2,Prdt_19KitKat,2].OffsetPlace.B=0
Ponto_STR[Pallet_2,Prdt_19KitKat,2].OffsetPlace.C=0
;ENDFOLD
;ENDFOLD

;FOLD PLACE 3
;FOLD PROPRIEDADES
Ponto_STR[Pallet_2,Prdt_19KitKat,3].NumCaixas = 1
Ponto_STR[Pallet_2,Prdt_19KitKat,3].PickOp = 6
Ponto_STR[Pallet_2,Prdt_19KitKat,3].ConfGarraOp = 0
Ponto_STR[Pallet_2,Prdt_19KitKat,3].FechaGarraOp = 0
Ponto_STR[Pallet_2,Prdt_19KitKat,3].AbreGarraOp = 0
Ponto_STR[Pallet_2,Prdt_19KitKat,3].SensoresCaixa = 6
Ponto_STR[Pallet_2,Prdt_19KitKat,3].TravaGarra = False
Ponto_STR[Pallet_2,Prdt_19KitKat,3].SkipGoHome = False
Ponto_STR[Pallet_2,Prdt_19KitKat,3].SkipSobeRelativo = False
Ponto_STR[Pallet_2,Prdt_19KitKat,3].XApp1Place=P2_19KitKat_3_App1
Ponto_STR[Pallet_2,Prdt_19KitKat,3].XApp2Place=P2_19KitKat_3_App2
Ponto_STR[Pallet_2,Prdt_19KitKat,3].XPlace=P2_19KitKat_3_Place
;ENDFOLD
;FOLD OffsetPlace
Ponto_STR[Pallet_2,Prdt_19KitKat,3].OffsetPlace.X=0
Ponto_STR[Pallet_2,Prdt_19KitKat,3].OffsetPlace.Y=0
Ponto_STR[Pallet_2,Prdt_19KitKat,3].OffsetPlace.Z=0
Ponto_STR[Pallet_2,Prdt_19KitKat,3].OffsetPlace.A=0
Ponto_STR[Pallet_2,Prdt_19KitKat,3].OffsetPlace.B=0
Ponto_STR[Pallet_2,Prdt_19KitKat,3].OffsetPlace.C=0
;ENDFOLD
;ENDFOLD

;FOLD PLACE 4
;FOLD PROPRIEDADES
Ponto_STR[Pallet_2,Prdt_19KitKat,4].NumCaixas = 4
Ponto_STR[Pallet_2,Prdt_19KitKat,4].PickOp = 1
Ponto_STR[Pallet_2,Prdt_19KitKat,4].ConfGarraOp = 0
Ponto_STR[Pallet_2,Prdt_19KitKat,4].FechaGarraOp = 0
Ponto_STR[Pallet_2,Prdt_19KitKat,4].AbreGarraOp = 0
Ponto_STR[Pallet_2,Prdt_19KitKat,4].SensoresCaixa = 12345
Ponto_STR[Pallet_2,Prdt_19KitKat,4].TravaGarra = False
Ponto_STR[Pallet_2,Prdt_19KitKat,4].SkipGoHome = False
Ponto_STR[Pallet_2,Prdt_19KitKat,4].SkipSobeRelativo = False
Ponto_STR[Pallet_2,Prdt_19KitKat,4].XApp1Place=P2_19KitKat_4_App1
Ponto_STR[Pallet_2,Prdt_19KitKat,4].XApp2Place=P2_19KitKat_4_App2
Ponto_STR[Pallet_2,Prdt_19KitKat,4].XPlace=P2_19KitKat_4_Place
;ENDFOLD
;FOLD OffsetPlace
Ponto_STR[Pallet_2,Prdt_19KitKat,4].OffsetPlace.X=0
Ponto_STR[Pallet_2,Prdt_19KitKat,4].OffsetPlace.Y=0
Ponto_STR[Pallet_2,Prdt_19KitKat,4].OffsetPlace.Z=0
Ponto_STR[Pallet_2,Prdt_19KitKat,4].OffsetPlace.A=0
Ponto_STR[Pallet_2,Prdt_19KitKat,4].OffsetPlace.B=0
Ponto_STR[Pallet_2,Prdt_19KitKat,4].OffsetPlace.C=0
;ENDFOLD
;ENDFOLD

;FOLD PLACE 5
;FOLD PROPRIEDADES
Ponto_STR[Pallet_2,Prdt_19KitKat,5].NumCaixas = 4
Ponto_STR[Pallet_2,Prdt_19KitKat,5].PickOp = 1
Ponto_STR[Pallet_2,Prdt_19KitKat,5].ConfGarraOp = 0
Ponto_STR[Pallet_2,Prdt_19KitKat,5].FechaGarraOp = 0
Ponto_STR[Pallet_2,Prdt_19KitKat,5].AbreGarraOp = 0
Ponto_STR[Pallet_2,Prdt_19KitKat,5].SensoresCaixa = 12345
Ponto_STR[Pallet_2,Prdt_19KitKat,5].TravaGarra = False
Ponto_STR[Pallet_2,Prdt_19KitKat,5].SkipGoHome = False
Ponto_STR[Pallet_2,Prdt_19KitKat,5].SkipSobeRelativo = False
Ponto_STR[Pallet_2,Prdt_19KitKat,5].XApp1Place=P2_19KitKat_5_App1
Ponto_STR[Pallet_2,Prdt_19KitKat,5].XApp2Place=P2_19KitKat_5_App2
Ponto_STR[Pallet_2,Prdt_19KitKat,5].XPlace=P2_19KitKat_5_Place
;ENDFOLD
;FOLD OffsetPlace
Ponto_STR[Pallet_2,Prdt_19KitKat,5].OffsetPlace.X=0
Ponto_STR[Pallet_2,Prdt_19KitKat,5].OffsetPlace.Y=0
Ponto_STR[Pallet_2,Prdt_19KitKat,5].OffsetPlace.Z=0
Ponto_STR[Pallet_2,Prdt_19KitKat,5].OffsetPlace.A=0
Ponto_STR[Pallet_2,Prdt_19KitKat,5].OffsetPlace.B=0
Ponto_STR[Pallet_2,Prdt_19KitKat,5].OffsetPlace.C=0
;ENDFOLD
;ENDFOLD

;FOLD PLACE 6
;FOLD PROPRIEDADES
Ponto_STR[Pallet_2,Prdt_19KitKat,6].NumCaixas = 4
Ponto_STR[Pallet_2,Prdt_19KitKat,6].PickOp = 1
Ponto_STR[Pallet_2,Prdt_19KitKat,6].ConfGarraOp = 0
Ponto_STR[Pallet_2,Prdt_19KitKat,6].FechaGarraOp = 0
Ponto_STR[Pallet_2,Prdt_19KitKat,6].AbreGarraOp = 0
Ponto_STR[Pallet_2,Prdt_19KitKat,6].SensoresCaixa = 12345
Ponto_STR[Pallet_2,Prdt_19KitKat,6].TravaGarra = False
Ponto_STR[Pallet_2,Prdt_19KitKat,6].SkipGoHome = False
Ponto_STR[Pallet_2,Prdt_19KitKat,6].SkipSobeRelativo = False
Ponto_STR[Pallet_2,Prdt_19KitKat,6].XApp1Place=P2_19KitKat_6_App1
Ponto_STR[Pallet_2,Prdt_19KitKat,6].XApp2Place=P2_19KitKat_6_App2
Ponto_STR[Pallet_2,Prdt_19KitKat,6].XPlace=P2_19KitKat_6_Place
;ENDFOLD
;FOLD OffsetPlace
Ponto_STR[Pallet_2,Prdt_19KitKat,6].OffsetPlace.X=0
Ponto_STR[Pallet_2,Prdt_19KitKat,6].OffsetPlace.Y=0
Ponto_STR[Pallet_2,Prdt_19KitKat,6].OffsetPlace.Z=0
Ponto_STR[Pallet_2,Prdt_19KitKat,6].OffsetPlace.A=0
Ponto_STR[Pallet_2,Prdt_19KitKat,6].OffsetPlace.B=0
Ponto_STR[Pallet_2,Prdt_19KitKat,6].OffsetPlace.C=0
;ENDFOLD
;ENDFOLD

;ENDFOLD
;FOLD LAYER 2: PLACE 7 ate 12
;FOLD PLACE 7
;FOLD PROPRIEDADES
Ponto_STR[Pallet_2,Prdt_19KitKat,7].NumCaixas = 1
Ponto_STR[Pallet_2,Prdt_19KitKat,7].PickOp = 1
Ponto_STR[Pallet_2,Prdt_19KitKat,7].ConfGarraOp = 0
Ponto_STR[Pallet_2,Prdt_19KitKat,7].FechaGarraOp = 0
Ponto_STR[Pallet_2,Prdt_19KitKat,7].AbreGarraOp = 0
Ponto_STR[Pallet_2,Prdt_19KitKat,7].SensoresCaixa = 1
Ponto_STR[Pallet_2,Prdt_19KitKat,7].TravaGarra = False
Ponto_STR[Pallet_2,Prdt_19KitKat,7].SkipGoHome = False
Ponto_STR[Pallet_2,Prdt_19KitKat,7].SkipSobeRelativo = False
Ponto_STR[Pallet_2,Prdt_19KitKat,7].XApp1Place=P2_19KitKat_7_App1
Ponto_STR[Pallet_2,Prdt_19KitKat,7].XApp2Place=P2_19KitKat_7_App2
Ponto_STR[Pallet_2,Prdt_19KitKat,7].XPlace=P2_19KitKat_7_Place
;ENDFOLD
;FOLD OffsetPlace
Ponto_STR[Pallet_2,Prdt_19KitKat,7].OffsetPlace.X=0
Ponto_STR[Pallet_2,Prdt_19KitKat,7].OffsetPlace.Y=0
Ponto_STR[Pallet_2,Prdt_19KitKat,7].OffsetPlace.Z=0
Ponto_STR[Pallet_2,Prdt_19KitKat,7].OffsetPlace.A=0
Ponto_STR[Pallet_2,Prdt_19KitKat,7].OffsetPlace.B=0
Ponto_STR[Pallet_2,Prdt_19KitKat,7].OffsetPlace.C=0
;ENDFOLD
;ENDFOLD

;FOLD PLACE 8
;FOLD PROPRIEDADES
Ponto_STR[Pallet_2,Prdt_19KitKat,8].NumCaixas = 1
Ponto_STR[Pallet_2,Prdt_19KitKat,8].PickOp = 1
Ponto_STR[Pallet_2,Prdt_19KitKat,8].ConfGarraOp = 0
Ponto_STR[Pallet_2,Prdt_19KitKat,8].FechaGarraOp = 0
Ponto_STR[Pallet_2,Prdt_19KitKat,8].AbreGarraOp = 0
Ponto_STR[Pallet_2,Prdt_19KitKat,8].SensoresCaixa = 1
Ponto_STR[Pallet_2,Prdt_19KitKat,8].TravaGarra = False
Ponto_STR[Pallet_2,Prdt_19KitKat,8].SkipGoHome = False
Ponto_STR[Pallet_2,Prdt_19KitKat,8].SkipSobeRelativo = False
Ponto_STR[Pallet_2,Prdt_19KitKat,8].XApp1Place=P2_19KitKat_8_App1
Ponto_STR[Pallet_2,Prdt_19KitKat,8].XApp2Place=P2_19KitKat_8_App2
Ponto_STR[Pallet_2,Prdt_19KitKat,8].XPlace=P2_19KitKat_8_Place
;ENDFOLD
;FOLD OffsetPlace
Ponto_STR[Pallet_2,Prdt_19KitKat,8].OffsetPlace.X=0
Ponto_STR[Pallet_2,Prdt_19KitKat,8].OffsetPlace.Y=0
Ponto_STR[Pallet_2,Prdt_19KitKat,8].OffsetPlace.Z=0
Ponto_STR[Pallet_2,Prdt_19KitKat,8].OffsetPlace.A=0
Ponto_STR[Pallet_2,Prdt_19KitKat,8].OffsetPlace.B=0
Ponto_STR[Pallet_2,Prdt_19KitKat,8].OffsetPlace.C=0
;ENDFOLD
;ENDFOLD

;FOLD PLACE 9
;FOLD PROPRIEDADES
Ponto_STR[Pallet_2,Prdt_19KitKat,9].NumCaixas = 1
Ponto_STR[Pallet_2,Prdt_19KitKat,9].PickOp = 1
Ponto_STR[Pallet_2,Prdt_19KitKat,9].ConfGarraOp = 0
Ponto_STR[Pallet_2,Prdt_19KitKat,9].FechaGarraOp = 0
Ponto_STR[Pallet_2,Prdt_19KitKat,9].AbreGarraOp = 0
Ponto_STR[Pallet_2,Prdt_19KitKat,9].SensoresCaixa = 1
Ponto_STR[Pallet_2,Prdt_19KitKat,9].TravaGarra = False
Ponto_STR[Pallet_2,Prdt_19KitKat,9].SkipGoHome = False
Ponto_STR[Pallet_2,Prdt_19KitKat,9].SkipSobeRelativo = False
Ponto_STR[Pallet_2,Prdt_19KitKat,9].XApp1Place=P2_19KitKat_9_App1
Ponto_STR[Pallet_2,Prdt_19KitKat,9].XApp2Place=P2_19KitKat_9_App2
Ponto_STR[Pallet_2,Prdt_19KitKat,9].XPlace=P2_19KitKat_9_Place
;ENDFOLD
;FOLD OffsetPlace
Ponto_STR[Pallet_2,Prdt_19KitKat,9].OffsetPlace.X=0
Ponto_STR[Pallet_2,Prdt_19KitKat,9].OffsetPlace.Y=0
Ponto_STR[Pallet_2,Prdt_19KitKat,9].OffsetPlace.Z=0
Ponto_STR[Pallet_2,Prdt_19KitKat,9].OffsetPlace.A=0
Ponto_STR[Pallet_2,Prdt_19KitKat,9].OffsetPlace.B=0
Ponto_STR[Pallet_2,Prdt_19KitKat,9].OffsetPlace.C=0
;ENDFOLD
;ENDFOLD

;FOLD PLACE 10
;FOLD PROPRIEDADES
Ponto_STR[Pallet_2,Prdt_19KitKat,10].NumCaixas = 4
Ponto_STR[Pallet_2,Prdt_19KitKat,10].PickOp = 1
Ponto_STR[Pallet_2,Prdt_19KitKat,10].ConfGarraOp = 0
Ponto_STR[Pallet_2,Prdt_19KitKat,10].FechaGarraOp = 0
Ponto_STR[Pallet_2,Prdt_19KitKat,10].AbreGarraOp = 1
Ponto_STR[Pallet_2,Prdt_19KitKat,10].SensoresCaixa = 12345
Ponto_STR[Pallet_2,Prdt_19KitKat,10].TravaGarra = True
Ponto_STR[Pallet_2,Prdt_19KitKat,10].SkipGoHome = False
Ponto_STR[Pallet_2,Prdt_19KitKat,10].SkipSobeRelativo = False
Ponto_STR[Pallet_2,Prdt_19KitKat,10].XApp1Place=P2_19KitKat_10_App1
Ponto_STR[Pallet_2,Prdt_19KitKat,10].XApp2Place=P2_19KitKat_10_App2
Ponto_STR[Pallet_2,Prdt_19KitKat,10].XPlace=P2_19KitKat_10_Place
;ENDFOLD
;FOLD OffsetPlace
Ponto_STR[Pallet_2,Prdt_19KitKat,10].OffsetPlace.X=0
Ponto_STR[Pallet_2,Prdt_19KitKat,10].OffsetPlace.Y=0
Ponto_STR[Pallet_2,Prdt_19KitKat,10].OffsetPlace.Z=0
Ponto_STR[Pallet_2,Prdt_19KitKat,10].OffsetPlace.A=0
Ponto_STR[Pallet_2,Prdt_19KitKat,10].OffsetPlace.B=0
Ponto_STR[Pallet_2,Prdt_19KitKat,10].OffsetPlace.C=0
;ENDFOLD
;ENDFOLD

;FOLD PLACE 11
;FOLD PROPRIEDADES
Ponto_STR[Pallet_2,Prdt_19KitKat,11].NumCaixas = 4
Ponto_STR[Pallet_2,Prdt_19KitKat,11].PickOp = 1
Ponto_STR[Pallet_2,Prdt_19KitKat,11].ConfGarraOp = 0
Ponto_STR[Pallet_2,Prdt_19KitKat,11].FechaGarraOp = 0
Ponto_STR[Pallet_2,Prdt_19KitKat,11].AbreGarraOp = 1
Ponto_STR[Pallet_2,Prdt_19KitKat,11].SensoresCaixa = 12345
Ponto_STR[Pallet_2,Prdt_19KitKat,11].TravaGarra = True
Ponto_STR[Pallet_2,Prdt_19KitKat,11].SkipGoHome = False
Ponto_STR[Pallet_2,Prdt_19KitKat,11].SkipSobeRelativo = False
Ponto_STR[Pallet_2,Prdt_19KitKat,11].XApp1Place=P2_19KitKat_11_App1
Ponto_STR[Pallet_2,Prdt_19KitKat,11].XApp2Place=P2_19KitKat_11_App2
Ponto_STR[Pallet_2,Prdt_19KitKat,11].XPlace=P2_19KitKat_11_Place
;ENDFOLD
;FOLD OffsetPlace
Ponto_STR[Pallet_2,Prdt_19KitKat,11].OffsetPlace.X=0
Ponto_STR[Pallet_2,Prdt_19KitKat,11].OffsetPlace.Y=0
Ponto_STR[Pallet_2,Prdt_19KitKat,11].OffsetPlace.Z=0
Ponto_STR[Pallet_2,Prdt_19KitKat,11].OffsetPlace.A=0
Ponto_STR[Pallet_2,Prdt_19KitKat,11].OffsetPlace.B=0
Ponto_STR[Pallet_2,Prdt_19KitKat,11].OffsetPlace.C=0
;ENDFOLD
;ENDFOLD

;FOLD PLACE 12
;FOLD PROPRIEDADES
Ponto_STR[Pallet_2,Prdt_19KitKat,12].NumCaixas = 4
Ponto_STR[Pallet_2,Prdt_19KitKat,12].PickOp = 1
Ponto_STR[Pallet_2,Prdt_19KitKat,12].ConfGarraOp = 0
Ponto_STR[Pallet_2,Prdt_19KitKat,12].FechaGarraOp = 0
Ponto_STR[Pallet_2,Prdt_19KitKat,12].AbreGarraOp = 1
Ponto_STR[Pallet_2,Prdt_19KitKat,12].SensoresCaixa = 12345
Ponto_STR[Pallet_2,Prdt_19KitKat,12].TravaGarra = True
Ponto_STR[Pallet_2,Prdt_19KitKat,12].SkipGoHome = False
Ponto_STR[Pallet_2,Prdt_19KitKat,12].SkipSobeRelativo = False
Ponto_STR[Pallet_2,Prdt_19KitKat,12].XApp1Place=P2_19KitKat_12_App1
Ponto_STR[Pallet_2,Prdt_19KitKat,12].XApp2Place=P2_19KitKat_12_App2
Ponto_STR[Pallet_2,Prdt_19KitKat,12].XPlace=P2_19KitKat_12_Place
;ENDFOLD
;FOLD OffsetPlace
Ponto_STR[Pallet_2,Prdt_19KitKat,12].OffsetPlace.X=0
Ponto_STR[Pallet_2,Prdt_19KitKat,12].OffsetPlace.Y=0
Ponto_STR[Pallet_2,Prdt_19KitKat,12].OffsetPlace.Z=0
Ponto_STR[Pallet_2,Prdt_19KitKat,12].OffsetPlace.A=0
Ponto_STR[Pallet_2,Prdt_19KitKat,12].OffsetPlace.B=0
Ponto_STR[Pallet_2,Prdt_19KitKat,12].OffsetPlace.C=0
;ENDFOLD
;ENDFOLD

;ENDFOLD
;ENDFOLD

;FOLD Pallet 2 - Produto 7Aero
;FOLD LAYER 1: PLACE 1 ate 8
;FOLD PLACE 1
;FOLD PROPRIEDADES
Ponto_STR[Pallet_2,Prdt_7Aero,1].NumCaixas = 3
Ponto_STR[Pallet_2,Prdt_7Aero,1].PickOp = 6
Ponto_STR[Pallet_2,Prdt_7Aero,1].ConfGarraOp = 0
Ponto_STR[Pallet_2,Prdt_7Aero,1].FechaGarraOp = 0
Ponto_STR[Pallet_2,Prdt_7Aero,1].AbreGarraOp = 0
Ponto_STR[Pallet_2,Prdt_7Aero,1].SensoresCaixa = 564
Ponto_STR[Pallet_2,Prdt_7Aero,1].TravaGarra = False
Ponto_STR[Pallet_2,Prdt_7Aero,1].SkipGoHome = False
Ponto_STR[Pallet_2,Prdt_7Aero,1].SkipSobeRelativo = False
Ponto_STR[Pallet_2,Prdt_7Aero,1].XApp1Place=P2_7Aero_1_App1
Ponto_STR[Pallet_2,Prdt_7Aero,1].XApp2Place=P2_7Aero_1_App2
Ponto_STR[Pallet_2,Prdt_7Aero,1].XPlace=P2_7Aero_1_Place
;ENDFOLD
;FOLD OffsetPlace
Ponto_STR[Pallet_2,Prdt_7Aero,1].OffsetPlace.X=0
Ponto_STR[Pallet_2,Prdt_7Aero,1].OffsetPlace.Y=0
Ponto_STR[Pallet_2,Prdt_7Aero,1].OffsetPlace.Z=0
Ponto_STR[Pallet_2,Prdt_7Aero,1].OffsetPlace.A=0
Ponto_STR[Pallet_2,Prdt_7Aero,1].OffsetPlace.B=0
Ponto_STR[Pallet_2,Prdt_7Aero,1].OffsetPlace.C=0
;ENDFOLD
;ENDFOLD

;FOLD PLACE 2
;FOLD PROPRIEDADES
Ponto_STR[Pallet_2,Prdt_7Aero,2].NumCaixas = 3
Ponto_STR[Pallet_2,Prdt_7Aero,2].PickOp = 6
Ponto_STR[Pallet_2,Prdt_7Aero,2].ConfGarraOp = 0
Ponto_STR[Pallet_2,Prdt_7Aero,2].FechaGarraOp = 0
Ponto_STR[Pallet_2,Prdt_7Aero,2].AbreGarraOp = 0
Ponto_STR[Pallet_2,Prdt_7Aero,2].SensoresCaixa = 564
Ponto_STR[Pallet_2,Prdt_7Aero,2].TravaGarra = False
Ponto_STR[Pallet_2,Prdt_7Aero,2].SkipGoHome = False
Ponto_STR[Pallet_2,Prdt_7Aero,2].SkipSobeRelativo = False
Ponto_STR[Pallet_2,Prdt_7Aero,2].XApp1Place=P2_7Aero_2_App1
Ponto_STR[Pallet_2,Prdt_7Aero,2].XApp2Place=P2_7Aero_2_App2
Ponto_STR[Pallet_2,Prdt_7Aero,2].XPlace=P2_7Aero_2_Place
;ENDFOLD
;FOLD OffsetPlace
Ponto_STR[Pallet_2,Prdt_7Aero,2].OffsetPlace.X=0
Ponto_STR[Pallet_2,Prdt_7Aero,2].OffsetPlace.Y=0
Ponto_STR[Pallet_2,Prdt_7Aero,2].OffsetPlace.Z=0
Ponto_STR[Pallet_2,Prdt_7Aero,2].OffsetPlace.A=0
Ponto_STR[Pallet_2,Prdt_7Aero,2].OffsetPlace.B=0
Ponto_STR[Pallet_2,Prdt_7Aero,2].OffsetPlace.C=0
;ENDFOLD
;ENDFOLD

;FOLD PLACE 3
;FOLD PROPRIEDADES
Ponto_STR[Pallet_2,Prdt_7Aero,3].NumCaixas = 2
Ponto_STR[Pallet_2,Prdt_7Aero,3].PickOp = 8
Ponto_STR[Pallet_2,Prdt_7Aero,3].ConfGarraOp = 5
Ponto_STR[Pallet_2,Prdt_7Aero,3].FechaGarraOp = 0
Ponto_STR[Pallet_2,Prdt_7Aero,3].AbreGarraOp = 0
Ponto_STR[Pallet_2,Prdt_7Aero,3].SensoresCaixa = 12
Ponto_STR[Pallet_2,Prdt_7Aero,3].TravaGarra = False
Ponto_STR[Pallet_2,Prdt_7Aero,3].SkipGoHome = False
Ponto_STR[Pallet_2,Prdt_7Aero,3].SkipSobeRelativo = False
Ponto_STR[Pallet_2,Prdt_7Aero,3].XApp1Place=P2_7Aero_3_App1
Ponto_STR[Pallet_2,Prdt_7Aero,3].XApp2Place=P2_7Aero_3_App2
Ponto_STR[Pallet_2,Prdt_7Aero,3].XPlace=P2_7Aero_3_Place
;ENDFOLD
;FOLD OffsetPlace
Ponto_STR[Pallet_2,Prdt_7Aero,3].OffsetPlace.X=0
Ponto_STR[Pallet_2,Prdt_7Aero,3].OffsetPlace.Y=0
Ponto_STR[Pallet_2,Prdt_7Aero,3].OffsetPlace.Z=0
Ponto_STR[Pallet_2,Prdt_7Aero,3].OffsetPlace.A=0
Ponto_STR[Pallet_2,Prdt_7Aero,3].OffsetPlace.B=0
Ponto_STR[Pallet_2,Prdt_7Aero,3].OffsetPlace.C=0
;ENDFOLD
;ENDFOLD

;FOLD PLACE 4
;FOLD PROPRIEDADES
Ponto_STR[Pallet_2,Prdt_7Aero,4].NumCaixas = 2
Ponto_STR[Pallet_2,Prdt_7Aero,4].PickOp = 8
Ponto_STR[Pallet_2,Prdt_7Aero,4].ConfGarraOp = 5
Ponto_STR[Pallet_2,Prdt_7Aero,4].FechaGarraOp = 0
Ponto_STR[Pallet_2,Prdt_7Aero,4].AbreGarraOp = 0
Ponto_STR[Pallet_2,Prdt_7Aero,4].SensoresCaixa = 12
Ponto_STR[Pallet_2,Prdt_7Aero,4].TravaGarra = False
Ponto_STR[Pallet_2,Prdt_7Aero,4].SkipGoHome = False
Ponto_STR[Pallet_2,Prdt_7Aero,4].SkipSobeRelativo = False
Ponto_STR[Pallet_2,Prdt_7Aero,4].XApp1Place=P2_7Aero_4_App1
Ponto_STR[Pallet_2,Prdt_7Aero,4].XApp2Place=P2_7Aero_4_App2
Ponto_STR[Pallet_2,Prdt_7Aero,4].XPlace=P2_7Aero_4_Place
;ENDFOLD
;FOLD OffsetPlace
Ponto_STR[Pallet_2,Prdt_7Aero,4].OffsetPlace.X=0
Ponto_STR[Pallet_2,Prdt_7Aero,4].OffsetPlace.Y=0
Ponto_STR[Pallet_2,Prdt_7Aero,4].OffsetPlace.Z=0
Ponto_STR[Pallet_2,Prdt_7Aero,4].OffsetPlace.A=0
Ponto_STR[Pallet_2,Prdt_7Aero,4].OffsetPlace.B=0
Ponto_STR[Pallet_2,Prdt_7Aero,4].OffsetPlace.C=0
;ENDFOLD
;ENDFOLD

;FOLD PLACE 5
;FOLD PROPRIEDADES
Ponto_STR[Pallet_2,Prdt_7Aero,5].NumCaixas = 3
Ponto_STR[Pallet_2,Prdt_7Aero,5].PickOp = 8
Ponto_STR[Pallet_2,Prdt_7Aero,5].ConfGarraOp = 5
Ponto_STR[Pallet_2,Prdt_7Aero,5].FechaGarraOp = 0
Ponto_STR[Pallet_2,Prdt_7Aero,5].AbreGarraOp = 1
Ponto_STR[Pallet_2,Prdt_7Aero,5].SensoresCaixa = 123
Ponto_STR[Pallet_2,Prdt_7Aero,5].TravaGarra = True
Ponto_STR[Pallet_2,Prdt_7Aero,5].SkipGoHome = False
Ponto_STR[Pallet_2,Prdt_7Aero,5].SkipSobeRelativo = False
Ponto_STR[Pallet_2,Prdt_7Aero,5].XApp1Place=P2_7Aero_5_App1
Ponto_STR[Pallet_2,Prdt_7Aero,5].XApp2Place=P2_7Aero_5_App2
Ponto_STR[Pallet_2,Prdt_7Aero,5].XPlace=P2_7Aero_5_Place
;ENDFOLD
;FOLD OffsetPlace
Ponto_STR[Pallet_2,Prdt_7Aero,5].OffsetPlace.X=0
Ponto_STR[Pallet_2,Prdt_7Aero,5].OffsetPlace.Y=0
Ponto_STR[Pallet_2,Prdt_7Aero,5].OffsetPlace.Z=0
Ponto_STR[Pallet_2,Prdt_7Aero,5].OffsetPlace.A=0
Ponto_STR[Pallet_2,Prdt_7Aero,5].OffsetPlace.B=0
Ponto_STR[Pallet_2,Prdt_7Aero,5].OffsetPlace.C=0
;ENDFOLD
;ENDFOLD

;FOLD PLACE 6
;FOLD PROPRIEDADES
Ponto_STR[Pallet_2,Prdt_7Aero,6].NumCaixas = 3
Ponto_STR[Pallet_2,Prdt_7Aero,6].PickOp = 8
Ponto_STR[Pallet_2,Prdt_7Aero,6].ConfGarraOp = 5
Ponto_STR[Pallet_2,Prdt_7Aero,6].FechaGarraOp = 0
Ponto_STR[Pallet_2,Prdt_7Aero,6].AbreGarraOp = 1
Ponto_STR[Pallet_2,Prdt_7Aero,6].SensoresCaixa = 123
Ponto_STR[Pallet_2,Prdt_7Aero,6].TravaGarra = True
Ponto_STR[Pallet_2,Prdt_7Aero,6].SkipGoHome = False
Ponto_STR[Pallet_2,Prdt_7Aero,6].SkipSobeRelativo = False
Ponto_STR[Pallet_2,Prdt_7Aero,6].XApp1Place=P2_7Aero_6_App1
Ponto_STR[Pallet_2,Prdt_7Aero,6].XApp2Place=P2_7Aero_6_App2
Ponto_STR[Pallet_2,Prdt_7Aero,6].XPlace=P2_7Aero_6_Place
;ENDFOLD
;FOLD OffsetPlace
Ponto_STR[Pallet_2,Prdt_7Aero,6].OffsetPlace.X=0
Ponto_STR[Pallet_2,Prdt_7Aero,6].OffsetPlace.Y=0
Ponto_STR[Pallet_2,Prdt_7Aero,6].OffsetPlace.Z=0
Ponto_STR[Pallet_2,Prdt_7Aero,6].OffsetPlace.A=0
Ponto_STR[Pallet_2,Prdt_7Aero,6].OffsetPlace.B=0
Ponto_STR[Pallet_2,Prdt_7Aero,6].OffsetPlace.C=0
;ENDFOLD
;ENDFOLD

;FOLD PLACE 7
;FOLD PROPRIEDADES
Ponto_STR[Pallet_2,Prdt_7Aero,7].NumCaixas = 2
Ponto_STR[Pallet_2,Prdt_7Aero,7].PickOp = 8
Ponto_STR[Pallet_2,Prdt_7Aero,7].ConfGarraOp = 5
Ponto_STR[Pallet_2,Prdt_7Aero,7].FechaGarraOp = 0
Ponto_STR[Pallet_2,Prdt_7Aero,7].AbreGarraOp = 1
Ponto_STR[Pallet_2,Prdt_7Aero,7].SensoresCaixa = 12
Ponto_STR[Pallet_2,Prdt_7Aero,7].TravaGarra = True
Ponto_STR[Pallet_2,Prdt_7Aero,7].SkipGoHome = False
Ponto_STR[Pallet_2,Prdt_7Aero,7].SkipSobeRelativo = False
Ponto_STR[Pallet_2,Prdt_7Aero,7].XApp1Place=P2_7Aero_7_App1
Ponto_STR[Pallet_2,Prdt_7Aero,7].XApp2Place=P2_7Aero_7_App2
Ponto_STR[Pallet_2,Prdt_7Aero,7].XPlace=P2_7Aero_7_Place
;ENDFOLD
;FOLD OffsetPlace
Ponto_STR[Pallet_2,Prdt_7Aero,7].OffsetPlace.X=0
Ponto_STR[Pallet_2,Prdt_7Aero,7].OffsetPlace.Y=0
Ponto_STR[Pallet_2,Prdt_7Aero,7].OffsetPlace.Z=0
Ponto_STR[Pallet_2,Prdt_7Aero,7].OffsetPlace.A=0
Ponto_STR[Pallet_2,Prdt_7Aero,7].OffsetPlace.B=0
Ponto_STR[Pallet_2,Prdt_7Aero,7].OffsetPlace.C=0
;ENDFOLD
;ENDFOLD

;FOLD PLACE 8
;FOLD PROPRIEDADES
Ponto_STR[Pallet_2,Prdt_7Aero,8].NumCaixas = 2
Ponto_STR[Pallet_2,Prdt_7Aero,8].PickOp = 8
Ponto_STR[Pallet_2,Prdt_7Aero,8].ConfGarraOp = 5
Ponto_STR[Pallet_2,Prdt_7Aero,8].FechaGarraOp = 0
Ponto_STR[Pallet_2,Prdt_7Aero,8].AbreGarraOp = 1
Ponto_STR[Pallet_2,Prdt_7Aero,8].SensoresCaixa = 12
Ponto_STR[Pallet_2,Prdt_7Aero,8].TravaGarra = True
Ponto_STR[Pallet_2,Prdt_7Aero,8].SkipGoHome = False
Ponto_STR[Pallet_2,Prdt_7Aero,8].SkipSobeRelativo = False
Ponto_STR[Pallet_2,Prdt_7Aero,8].XApp1Place=P2_7Aero_8_App1
Ponto_STR[Pallet_2,Prdt_7Aero,8].XApp2Place=P2_7Aero_8_App2
Ponto_STR[Pallet_2,Prdt_7Aero,8].XPlace=P2_7Aero_8_Place
;ENDFOLD
;FOLD OffsetPlace
Ponto_STR[Pallet_2,Prdt_7Aero,8].OffsetPlace.X=0
Ponto_STR[Pallet_2,Prdt_7Aero,8].OffsetPlace.Y=0
Ponto_STR[Pallet_2,Prdt_7Aero,8].OffsetPlace.Z=0
Ponto_STR[Pallet_2,Prdt_7Aero,8].OffsetPlace.A=0
Ponto_STR[Pallet_2,Prdt_7Aero,8].OffsetPlace.B=0
Ponto_STR[Pallet_2,Prdt_7Aero,8].OffsetPlace.C=0
;ENDFOLD
;ENDFOLD

;ENDFOLD
;FOLD LAYER 2: PLACE 9 ate 16
;FOLD PLACE 9
;FOLD PROPRIEDADES
Ponto_STR[Pallet_2,Prdt_7Aero,9].NumCaixas = 2
Ponto_STR[Pallet_2,Prdt_7Aero,9].PickOp = 8
Ponto_STR[Pallet_2,Prdt_7Aero,9].ConfGarraOp = 5
Ponto_STR[Pallet_2,Prdt_7Aero,9].FechaGarraOp = 0
Ponto_STR[Pallet_2,Prdt_7Aero,9].AbreGarraOp = 1
Ponto_STR[Pallet_2,Prdt_7Aero,9].SensoresCaixa = 12
Ponto_STR[Pallet_2,Prdt_7Aero,9].TravaGarra = True
Ponto_STR[Pallet_2,Prdt_7Aero,9].SkipGoHome = False
Ponto_STR[Pallet_2,Prdt_7Aero,9].SkipSobeRelativo = False
Ponto_STR[Pallet_2,Prdt_7Aero,9].XApp1Place=P2_7Aero_9_App1
Ponto_STR[Pallet_2,Prdt_7Aero,9].XApp2Place=P2_7Aero_9_App2
Ponto_STR[Pallet_2,Prdt_7Aero,9].XPlace=P2_7Aero_9_Place
;ENDFOLD
;FOLD OffsetPlace
Ponto_STR[Pallet_2,Prdt_7Aero,9].OffsetPlace.X=0
Ponto_STR[Pallet_2,Prdt_7Aero,9].OffsetPlace.Y=0
Ponto_STR[Pallet_2,Prdt_7Aero,9].OffsetPlace.Z=0
Ponto_STR[Pallet_2,Prdt_7Aero,9].OffsetPlace.A=0
Ponto_STR[Pallet_2,Prdt_7Aero,9].OffsetPlace.B=0
Ponto_STR[Pallet_2,Prdt_7Aero,9].OffsetPlace.C=0
;ENDFOLD
;ENDFOLD

;FOLD PLACE 10
;FOLD PROPRIEDADES
Ponto_STR[Pallet_2,Prdt_7Aero,10].NumCaixas = 2
Ponto_STR[Pallet_2,Prdt_7Aero,10].PickOp = 8
Ponto_STR[Pallet_2,Prdt_7Aero,10].ConfGarraOp = 5
Ponto_STR[Pallet_2,Prdt_7Aero,10].FechaGarraOp = 0
Ponto_STR[Pallet_2,Prdt_7Aero,10].AbreGarraOp = 1
Ponto_STR[Pallet_2,Prdt_7Aero,10].SensoresCaixa = 12
Ponto_STR[Pallet_2,Prdt_7Aero,10].TravaGarra = True
Ponto_STR[Pallet_2,Prdt_7Aero,10].SkipGoHome = False
Ponto_STR[Pallet_2,Prdt_7Aero,10].SkipSobeRelativo = False
Ponto_STR[Pallet_2,Prdt_7Aero,10].XApp1Place=P2_7Aero_10_App1
Ponto_STR[Pallet_2,Prdt_7Aero,10].XApp2Place=P2_7Aero_10_App2
Ponto_STR[Pallet_2,Prdt_7Aero,10].XPlace=P2_7Aero_10_Place
;ENDFOLD
;FOLD OffsetPlace
Ponto_STR[Pallet_2,Prdt_7Aero,10].OffsetPlace.X=0
Ponto_STR[Pallet_2,Prdt_7Aero,10].OffsetPlace.Y=0
Ponto_STR[Pallet_2,Prdt_7Aero,10].OffsetPlace.Z=0
Ponto_STR[Pallet_2,Prdt_7Aero,10].OffsetPlace.A=0
Ponto_STR[Pallet_2,Prdt_7Aero,10].OffsetPlace.B=0
Ponto_STR[Pallet_2,Prdt_7Aero,10].OffsetPlace.C=0
;ENDFOLD
;ENDFOLD

;FOLD PLACE 11
;FOLD PROPRIEDADES
Ponto_STR[Pallet_2,Prdt_7Aero,11].NumCaixas = 3
Ponto_STR[Pallet_2,Prdt_7Aero,11].PickOp = 8
Ponto_STR[Pallet_2,Prdt_7Aero,11].ConfGarraOp = 5
Ponto_STR[Pallet_2,Prdt_7Aero,11].FechaGarraOp = 0
Ponto_STR[Pallet_2,Prdt_7Aero,11].AbreGarraOp = 0
Ponto_STR[Pallet_2,Prdt_7Aero,11].SensoresCaixa = 123
Ponto_STR[Pallet_2,Prdt_7Aero,11].TravaGarra = False
Ponto_STR[Pallet_2,Prdt_7Aero,11].SkipGoHome = False
Ponto_STR[Pallet_2,Prdt_7Aero,11].SkipSobeRelativo = False
Ponto_STR[Pallet_2,Prdt_7Aero,11].XApp1Place=P2_7Aero_11_App1
Ponto_STR[Pallet_2,Prdt_7Aero,11].XApp2Place=P2_7Aero_11_App2
Ponto_STR[Pallet_2,Prdt_7Aero,11].XPlace=P2_7Aero_11_Place
;ENDFOLD
;FOLD OffsetPlace
Ponto_STR[Pallet_2,Prdt_7Aero,11].OffsetPlace.X=0
Ponto_STR[Pallet_2,Prdt_7Aero,11].OffsetPlace.Y=0
Ponto_STR[Pallet_2,Prdt_7Aero,11].OffsetPlace.Z=0
Ponto_STR[Pallet_2,Prdt_7Aero,11].OffsetPlace.A=0
Ponto_STR[Pallet_2,Prdt_7Aero,11].OffsetPlace.B=0
Ponto_STR[Pallet_2,Prdt_7Aero,11].OffsetPlace.C=0
;ENDFOLD
;ENDFOLD

;FOLD PLACE 12
;FOLD PROPRIEDADES
Ponto_STR[Pallet_2,Prdt_7Aero,12].NumCaixas = 3
Ponto_STR[Pallet_2,Prdt_7Aero,12].PickOp = 8
Ponto_STR[Pallet_2,Prdt_7Aero,12].ConfGarraOp = 5
Ponto_STR[Pallet_2,Prdt_7Aero,12].FechaGarraOp = 0
Ponto_STR[Pallet_2,Prdt_7Aero,12].AbreGarraOp = 0
Ponto_STR[Pallet_2,Prdt_7Aero,12].SensoresCaixa = 123
Ponto_STR[Pallet_2,Prdt_7Aero,12].TravaGarra = False
Ponto_STR[Pallet_2,Prdt_7Aero,12].SkipGoHome = False
Ponto_STR[Pallet_2,Prdt_7Aero,12].SkipSobeRelativo = False
Ponto_STR[Pallet_2,Prdt_7Aero,12].XApp1Place=P2_7Aero_12_App1
Ponto_STR[Pallet_2,Prdt_7Aero,12].XApp2Place=P2_7Aero_12_App2
Ponto_STR[Pallet_2,Prdt_7Aero,12].XPlace=P2_7Aero_12_Place
;ENDFOLD
;FOLD OffsetPlace
Ponto_STR[Pallet_2,Prdt_7Aero,12].OffsetPlace.X=0
Ponto_STR[Pallet_2,Prdt_7Aero,12].OffsetPlace.Y=0
Ponto_STR[Pallet_2,Prdt_7Aero,12].OffsetPlace.Z=0
Ponto_STR[Pallet_2,Prdt_7Aero,12].OffsetPlace.A=0
Ponto_STR[Pallet_2,Prdt_7Aero,12].OffsetPlace.B=0
Ponto_STR[Pallet_2,Prdt_7Aero,12].OffsetPlace.C=0
;ENDFOLD
;ENDFOLD

;FOLD PLACE 13
;FOLD PROPRIEDADES
Ponto_STR[Pallet_2,Prdt_7Aero,13].NumCaixas = 3
Ponto_STR[Pallet_2,Prdt_7Aero,13].PickOp = 8
Ponto_STR[Pallet_2,Prdt_7Aero,13].ConfGarraOp = 5
Ponto_STR[Pallet_2,Prdt_7Aero,13].FechaGarraOp = 0
Ponto_STR[Pallet_2,Prdt_7Aero,13].AbreGarraOp = 0
Ponto_STR[Pallet_2,Prdt_7Aero,13].SensoresCaixa = 123
Ponto_STR[Pallet_2,Prdt_7Aero,13].TravaGarra = False
Ponto_STR[Pallet_2,Prdt_7Aero,13].SkipGoHome = False
Ponto_STR[Pallet_2,Prdt_7Aero,13].SkipSobeRelativo = False
Ponto_STR[Pallet_2,Prdt_7Aero,13].XApp1Place=P2_7Aero_13_App1
Ponto_STR[Pallet_2,Prdt_7Aero,13].XApp2Place=P2_7Aero_13_App2
Ponto_STR[Pallet_2,Prdt_7Aero,13].XPlace=P2_7Aero_13_Place
;ENDFOLD
;FOLD OffsetPlace
Ponto_STR[Pallet_2,Prdt_7Aero,13].OffsetPlace.X=0
Ponto_STR[Pallet_2,Prdt_7Aero,13].OffsetPlace.Y=0
Ponto_STR[Pallet_2,Prdt_7Aero,13].OffsetPlace.Z=0
Ponto_STR[Pallet_2,Prdt_7Aero,13].OffsetPlace.A=0
Ponto_STR[Pallet_2,Prdt_7Aero,13].OffsetPlace.B=0
Ponto_STR[Pallet_2,Prdt_7Aero,13].OffsetPlace.C=0
;ENDFOLD
;ENDFOLD

;FOLD PLACE 14
;FOLD PROPRIEDADES
Ponto_STR[Pallet_2,Prdt_7Aero,14].NumCaixas = 3
Ponto_STR[Pallet_2,Prdt_7Aero,14].PickOp = 8
Ponto_STR[Pallet_2,Prdt_7Aero,14].ConfGarraOp = 5
Ponto_STR[Pallet_2,Prdt_7Aero,14].FechaGarraOp = 0
Ponto_STR[Pallet_2,Prdt_7Aero,14].AbreGarraOp = 0
Ponto_STR[Pallet_2,Prdt_7Aero,14].SensoresCaixa = 123
Ponto_STR[Pallet_2,Prdt_7Aero,14].TravaGarra = False
Ponto_STR[Pallet_2,Prdt_7Aero,14].SkipGoHome = False
Ponto_STR[Pallet_2,Prdt_7Aero,14].SkipSobeRelativo = False
Ponto_STR[Pallet_2,Prdt_7Aero,14].XApp1Place=P2_7Aero_14_App1
Ponto_STR[Pallet_2,Prdt_7Aero,14].XApp2Place=P2_7Aero_14_App2
Ponto_STR[Pallet_2,Prdt_7Aero,14].XPlace=P2_7Aero_14_Place
;ENDFOLD
;FOLD OffsetPlace
Ponto_STR[Pallet_2,Prdt_7Aero,14].OffsetPlace.X=0
Ponto_STR[Pallet_2,Prdt_7Aero,14].OffsetPlace.Y=0
Ponto_STR[Pallet_2,Prdt_7Aero,14].OffsetPlace.Z=0
Ponto_STR[Pallet_2,Prdt_7Aero,14].OffsetPlace.A=0
Ponto_STR[Pallet_2,Prdt_7Aero,14].OffsetPlace.B=0
Ponto_STR[Pallet_2,Prdt_7Aero,14].OffsetPlace.C=0
;ENDFOLD
;ENDFOLD

;FOLD PLACE 15
;FOLD PROPRIEDADES
Ponto_STR[Pallet_2,Prdt_7Aero,15].NumCaixas = 2
Ponto_STR[Pallet_2,Prdt_7Aero,15].PickOp = 8
Ponto_STR[Pallet_2,Prdt_7Aero,15].ConfGarraOp = 5
Ponto_STR[Pallet_2,Prdt_7Aero,15].FechaGarraOp = 0
Ponto_STR[Pallet_2,Prdt_7Aero,15].AbreGarraOp = 1
Ponto_STR[Pallet_2,Prdt_7Aero,15].SensoresCaixa = 12
Ponto_STR[Pallet_2,Prdt_7Aero,15].TravaGarra = True
Ponto_STR[Pallet_2,Prdt_7Aero,15].SkipGoHome = False
Ponto_STR[Pallet_2,Prdt_7Aero,15].SkipSobeRelativo = False
Ponto_STR[Pallet_2,Prdt_7Aero,15].XApp1Place=P2_7Aero_15_App1
Ponto_STR[Pallet_2,Prdt_7Aero,15].XApp2Place=P2_7Aero_15_App2
Ponto_STR[Pallet_2,Prdt_7Aero,15].XPlace=P2_7Aero_15_Place
;ENDFOLD
;FOLD OffsetPlace
Ponto_STR[Pallet_2,Prdt_7Aero,15].OffsetPlace.X=0
Ponto_STR[Pallet_2,Prdt_7Aero,15].OffsetPlace.Y=0
Ponto_STR[Pallet_2,Prdt_7Aero,15].OffsetPlace.Z=0
Ponto_STR[Pallet_2,Prdt_7Aero,15].OffsetPlace.A=0
Ponto_STR[Pallet_2,Prdt_7Aero,15].OffsetPlace.B=0
Ponto_STR[Pallet_2,Prdt_7Aero,15].OffsetPlace.C=0
;ENDFOLD
;ENDFOLD

;FOLD PLACE 16
;FOLD PROPRIEDADES
Ponto_STR[Pallet_2,Prdt_7Aero,16].NumCaixas = 2
Ponto_STR[Pallet_2,Prdt_7Aero,16].PickOp = 8
Ponto_STR[Pallet_2,Prdt_7Aero,16].ConfGarraOp = 5
Ponto_STR[Pallet_2,Prdt_7Aero,16].FechaGarraOp = 0
Ponto_STR[Pallet_2,Prdt_7Aero,16].AbreGarraOp = 1
Ponto_STR[Pallet_2,Prdt_7Aero,16].SensoresCaixa = 12
Ponto_STR[Pallet_2,Prdt_7Aero,16].TravaGarra = True
Ponto_STR[Pallet_2,Prdt_7Aero,16].SkipGoHome = False
Ponto_STR[Pallet_2,Prdt_7Aero,16].SkipSobeRelativo = False
Ponto_STR[Pallet_2,Prdt_7Aero,16].XApp1Place=P2_7Aero_16_App1
Ponto_STR[Pallet_2,Prdt_7Aero,16].XApp2Place=P2_7Aero_16_App2
Ponto_STR[Pallet_2,Prdt_7Aero,16].XPlace=P2_7Aero_16_Place
;ENDFOLD
;FOLD OffsetPlace
Ponto_STR[Pallet_2,Prdt_7Aero,16].OffsetPlace.X=0
Ponto_STR[Pallet_2,Prdt_7Aero,16].OffsetPlace.Y=0
Ponto_STR[Pallet_2,Prdt_7Aero,16].OffsetPlace.Z=0
Ponto_STR[Pallet_2,Prdt_7Aero,16].OffsetPlace.A=0
Ponto_STR[Pallet_2,Prdt_7Aero,16].OffsetPlace.B=0
Ponto_STR[Pallet_2,Prdt_7Aero,16].OffsetPlace.C=0
;ENDFOLD
;ENDFOLD

;ENDFOLD
;ENDFOLD

;FOLD Pallet 2 - Produto 15CoffeCrisp
;FOLD LAYER 1: PLACE 1 ate 7
;FOLD PLACE 1
;FOLD PROPRIEDADES
Ponto_STR[Pallet_2,Prdt_15CoffeCrisp,1].NumCaixas = 1
Ponto_STR[Pallet_2,Prdt_15CoffeCrisp,1].PickOp = 8
Ponto_STR[Pallet_2,Prdt_15CoffeCrisp,1].ConfGarraOp = 5
Ponto_STR[Pallet_2,Prdt_15CoffeCrisp,1].FechaGarraOp = 0
Ponto_STR[Pallet_2,Prdt_15CoffeCrisp,1].AbreGarraOp = 0
Ponto_STR[Pallet_2,Prdt_15CoffeCrisp,1].SensoresCaixa = 1
Ponto_STR[Pallet_2,Prdt_15CoffeCrisp,1].TravaGarra = False
Ponto_STR[Pallet_2,Prdt_15CoffeCrisp,1].SkipGoHome = False
Ponto_STR[Pallet_2,Prdt_15CoffeCrisp,1].SkipSobeRelativo = False
Ponto_STR[Pallet_2,Prdt_15CoffeCrisp,1].XApp1Place=P2_15CoffeCrisp_1_App1
Ponto_STR[Pallet_2,Prdt_15CoffeCrisp,1].XApp2Place=P2_15CoffeCrisp_1_App2
Ponto_STR[Pallet_2,Prdt_15CoffeCrisp,1].XPlace=P2_15CoffeCrisp_1_Place
;ENDFOLD
;FOLD OffsetPlace
Ponto_STR[Pallet_2,Prdt_15CoffeCrisp,1].OffsetPlace.X=0
Ponto_STR[Pallet_2,Prdt_15CoffeCrisp,1].OffsetPlace.Y=0
Ponto_STR[Pallet_2,Prdt_15CoffeCrisp,1].OffsetPlace.Z=0
Ponto_STR[Pallet_2,Prdt_15CoffeCrisp,1].OffsetPlace.A=0
Ponto_STR[Pallet_2,Prdt_15CoffeCrisp,1].OffsetPlace.B=0
Ponto_STR[Pallet_2,Prdt_15CoffeCrisp,1].OffsetPlace.C=0
;ENDFOLD
;ENDFOLD

;FOLD PLACE 2
;FOLD PROPRIEDADES
Ponto_STR[Pallet_2,Prdt_15CoffeCrisp,2].NumCaixas = 1
Ponto_STR[Pallet_2,Prdt_15CoffeCrisp,2].PickOp = 8
Ponto_STR[Pallet_2,Prdt_15CoffeCrisp,2].ConfGarraOp = 5
Ponto_STR[Pallet_2,Prdt_15CoffeCrisp,2].FechaGarraOp = 0
Ponto_STR[Pallet_2,Prdt_15CoffeCrisp,2].AbreGarraOp = 0
Ponto_STR[Pallet_2,Prdt_15CoffeCrisp,2].SensoresCaixa = 1
Ponto_STR[Pallet_2,Prdt_15CoffeCrisp,2].TravaGarra = False
Ponto_STR[Pallet_2,Prdt_15CoffeCrisp,2].SkipGoHome = False
Ponto_STR[Pallet_2,Prdt_15CoffeCrisp,2].SkipSobeRelativo = False
Ponto_STR[Pallet_2,Prdt_15CoffeCrisp,2].XApp1Place=P2_15CoffeCrisp_2_App1
Ponto_STR[Pallet_2,Prdt_15CoffeCrisp,2].XApp2Place=P2_15CoffeCrisp_2_App2
Ponto_STR[Pallet_2,Prdt_15CoffeCrisp,2].XPlace=P2_15CoffeCrisp_2_Place
;ENDFOLD
;FOLD OffsetPlace
Ponto_STR[Pallet_2,Prdt_15CoffeCrisp,2].OffsetPlace.X=0
Ponto_STR[Pallet_2,Prdt_15CoffeCrisp,2].OffsetPlace.Y=0
Ponto_STR[Pallet_2,Prdt_15CoffeCrisp,2].OffsetPlace.Z=0
Ponto_STR[Pallet_2,Prdt_15CoffeCrisp,2].OffsetPlace.A=0
Ponto_STR[Pallet_2,Prdt_15CoffeCrisp,2].OffsetPlace.B=0
Ponto_STR[Pallet_2,Prdt_15CoffeCrisp,2].OffsetPlace.C=0
;ENDFOLD
;ENDFOLD

;FOLD PLACE 3
;FOLD PROPRIEDADES
Ponto_STR[Pallet_2,Prdt_15CoffeCrisp,3].NumCaixas = 1
Ponto_STR[Pallet_2,Prdt_15CoffeCrisp,3].PickOp = 8
Ponto_STR[Pallet_2,Prdt_15CoffeCrisp,3].ConfGarraOp = 5
Ponto_STR[Pallet_2,Prdt_15CoffeCrisp,3].FechaGarraOp = 0
Ponto_STR[Pallet_2,Prdt_15CoffeCrisp,3].AbreGarraOp = 0
Ponto_STR[Pallet_2,Prdt_15CoffeCrisp,3].SensoresCaixa = 1
Ponto_STR[Pallet_2,Prdt_15CoffeCrisp,3].TravaGarra = False
Ponto_STR[Pallet_2,Prdt_15CoffeCrisp,3].SkipGoHome = False
Ponto_STR[Pallet_2,Prdt_15CoffeCrisp,3].SkipSobeRelativo = False
Ponto_STR[Pallet_2,Prdt_15CoffeCrisp,3].XApp1Place=P2_15CoffeCrisp_3_App1
Ponto_STR[Pallet_2,Prdt_15CoffeCrisp,3].XApp2Place=P2_15CoffeCrisp_3_App2
Ponto_STR[Pallet_2,Prdt_15CoffeCrisp,3].XPlace=P2_15CoffeCrisp_3_Place
;ENDFOLD
;FOLD OffsetPlace
Ponto_STR[Pallet_2,Prdt_15CoffeCrisp,3].OffsetPlace.X=0
Ponto_STR[Pallet_2,Prdt_15CoffeCrisp,3].OffsetPlace.Y=0
Ponto_STR[Pallet_2,Prdt_15CoffeCrisp,3].OffsetPlace.Z=0
Ponto_STR[Pallet_2,Prdt_15CoffeCrisp,3].OffsetPlace.A=0
Ponto_STR[Pallet_2,Prdt_15CoffeCrisp,3].OffsetPlace.B=0
Ponto_STR[Pallet_2,Prdt_15CoffeCrisp,3].OffsetPlace.C=0
;ENDFOLD
;ENDFOLD

;FOLD PLACE 4
;FOLD PROPRIEDADES
Ponto_STR[Pallet_2,Prdt_15CoffeCrisp,4].NumCaixas = 2
Ponto_STR[Pallet_2,Prdt_15CoffeCrisp,4].PickOp = 8
Ponto_STR[Pallet_2,Prdt_15CoffeCrisp,4].ConfGarraOp = 5
Ponto_STR[Pallet_2,Prdt_15CoffeCrisp,4].FechaGarraOp = 0
Ponto_STR[Pallet_2,Prdt_15CoffeCrisp,4].AbreGarraOp = 1
Ponto_STR[Pallet_2,Prdt_15CoffeCrisp,4].SensoresCaixa = 123
Ponto_STR[Pallet_2,Prdt_15CoffeCrisp,4].TravaGarra = True
Ponto_STR[Pallet_2,Prdt_15CoffeCrisp,4].SkipGoHome = False
Ponto_STR[Pallet_2,Prdt_15CoffeCrisp,4].SkipSobeRelativo = False
Ponto_STR[Pallet_2,Prdt_15CoffeCrisp,4].XApp1Place=P2_15CoffeCrisp_4_App1
Ponto_STR[Pallet_2,Prdt_15CoffeCrisp,4].XApp2Place=P2_15CoffeCrisp_4_App2
Ponto_STR[Pallet_2,Prdt_15CoffeCrisp,4].XPlace=P2_15CoffeCrisp_4_Place
;ENDFOLD
;FOLD OffsetPlace
Ponto_STR[Pallet_2,Prdt_15CoffeCrisp,4].OffsetPlace.X=0
Ponto_STR[Pallet_2,Prdt_15CoffeCrisp,4].OffsetPlace.Y=0
Ponto_STR[Pallet_2,Prdt_15CoffeCrisp,4].OffsetPlace.Z=0
Ponto_STR[Pallet_2,Prdt_15CoffeCrisp,4].OffsetPlace.A=0
Ponto_STR[Pallet_2,Prdt_15CoffeCrisp,4].OffsetPlace.B=0
Ponto_STR[Pallet_2,Prdt_15CoffeCrisp,4].OffsetPlace.C=0
;ENDFOLD
;ENDFOLD

;FOLD PLACE 5
;FOLD PROPRIEDADES
Ponto_STR[Pallet_2,Prdt_15CoffeCrisp,5].NumCaixas = 2
Ponto_STR[Pallet_2,Prdt_15CoffeCrisp,5].PickOp = 8
Ponto_STR[Pallet_2,Prdt_15CoffeCrisp,5].ConfGarraOp = 5
Ponto_STR[Pallet_2,Prdt_15CoffeCrisp,5].FechaGarraOp = 0
Ponto_STR[Pallet_2,Prdt_15CoffeCrisp,5].AbreGarraOp = 1
Ponto_STR[Pallet_2,Prdt_15CoffeCrisp,5].SensoresCaixa = 123
Ponto_STR[Pallet_2,Prdt_15CoffeCrisp,5].TravaGarra = True
Ponto_STR[Pallet_2,Prdt_15CoffeCrisp,5].SkipGoHome = False
Ponto_STR[Pallet_2,Prdt_15CoffeCrisp,5].SkipSobeRelativo = False
Ponto_STR[Pallet_2,Prdt_15CoffeCrisp,5].XApp1Place=P2_15CoffeCrisp_5_App1
Ponto_STR[Pallet_2,Prdt_15CoffeCrisp,5].XApp2Place=P2_15CoffeCrisp_5_App2
Ponto_STR[Pallet_2,Prdt_15CoffeCrisp,5].XPlace=P2_15CoffeCrisp_5_Place
;ENDFOLD
;FOLD OffsetPlace
Ponto_STR[Pallet_2,Prdt_15CoffeCrisp,5].OffsetPlace.X=0
Ponto_STR[Pallet_2,Prdt_15CoffeCrisp,5].OffsetPlace.Y=0
Ponto_STR[Pallet_2,Prdt_15CoffeCrisp,5].OffsetPlace.Z=0
Ponto_STR[Pallet_2,Prdt_15CoffeCrisp,5].OffsetPlace.A=0
Ponto_STR[Pallet_2,Prdt_15CoffeCrisp,5].OffsetPlace.B=0
Ponto_STR[Pallet_2,Prdt_15CoffeCrisp,5].OffsetPlace.C=0
;ENDFOLD
;ENDFOLD

;FOLD PLACE 6
;FOLD PROPRIEDADES
Ponto_STR[Pallet_2,Prdt_15CoffeCrisp,6].NumCaixas = 3
Ponto_STR[Pallet_2,Prdt_15CoffeCrisp,6].PickOp = 8
Ponto_STR[Pallet_2,Prdt_15CoffeCrisp,6].ConfGarraOp = 5
Ponto_STR[Pallet_2,Prdt_15CoffeCrisp,6].FechaGarraOp = 0
Ponto_STR[Pallet_2,Prdt_15CoffeCrisp,6].AbreGarraOp = 0
Ponto_STR[Pallet_2,Prdt_15CoffeCrisp,6].SensoresCaixa = 1234
Ponto_STR[Pallet_2,Prdt_15CoffeCrisp,6].TravaGarra = False
Ponto_STR[Pallet_2,Prdt_15CoffeCrisp,6].SkipGoHome = False
Ponto_STR[Pallet_2,Prdt_15CoffeCrisp,6].SkipSobeRelativo = False
Ponto_STR[Pallet_2,Prdt_15CoffeCrisp,6].XApp1Place=P2_15CoffeCrisp_6_App1
Ponto_STR[Pallet_2,Prdt_15CoffeCrisp,6].XApp2Place=P2_15CoffeCrisp_6_App2
Ponto_STR[Pallet_2,Prdt_15CoffeCrisp,6].XPlace=P2_15CoffeCrisp_6_Place
;ENDFOLD
;FOLD OffsetPlace
Ponto_STR[Pallet_2,Prdt_15CoffeCrisp,6].OffsetPlace.X=0
Ponto_STR[Pallet_2,Prdt_15CoffeCrisp,6].OffsetPlace.Y=0
Ponto_STR[Pallet_2,Prdt_15CoffeCrisp,6].OffsetPlace.Z=0
Ponto_STR[Pallet_2,Prdt_15CoffeCrisp,6].OffsetPlace.A=0
Ponto_STR[Pallet_2,Prdt_15CoffeCrisp,6].OffsetPlace.B=0
Ponto_STR[Pallet_2,Prdt_15CoffeCrisp,6].OffsetPlace.C=0
;ENDFOLD
;ENDFOLD

;FOLD PLACE 7
;FOLD PROPRIEDADES
Ponto_STR[Pallet_2,Prdt_15CoffeCrisp,7].NumCaixas = 3
Ponto_STR[Pallet_2,Prdt_15CoffeCrisp,7].PickOp = 8
Ponto_STR[Pallet_2,Prdt_15CoffeCrisp,7].ConfGarraOp = 5
Ponto_STR[Pallet_2,Prdt_15CoffeCrisp,7].FechaGarraOp = 0
Ponto_STR[Pallet_2,Prdt_15CoffeCrisp,7].AbreGarraOp = 0
Ponto_STR[Pallet_2,Prdt_15CoffeCrisp,7].SensoresCaixa = 1234
Ponto_STR[Pallet_2,Prdt_15CoffeCrisp,7].TravaGarra = False
Ponto_STR[Pallet_2,Prdt_15CoffeCrisp,7].SkipGoHome = False
Ponto_STR[Pallet_2,Prdt_15CoffeCrisp,7].SkipSobeRelativo = False
Ponto_STR[Pallet_2,Prdt_15CoffeCrisp,7].XApp1Place=P2_15CoffeCrisp_7_App1
Ponto_STR[Pallet_2,Prdt_15CoffeCrisp,7].XApp2Place=P2_15CoffeCrisp_7_App2
Ponto_STR[Pallet_2,Prdt_15CoffeCrisp,7].XPlace=P2_15CoffeCrisp_7_Place
;ENDFOLD
;FOLD OffsetPlace
Ponto_STR[Pallet_2,Prdt_15CoffeCrisp,7].OffsetPlace.X=0
Ponto_STR[Pallet_2,Prdt_15CoffeCrisp,7].OffsetPlace.Y=0
Ponto_STR[Pallet_2,Prdt_15CoffeCrisp,7].OffsetPlace.Z=0
Ponto_STR[Pallet_2,Prdt_15CoffeCrisp,7].OffsetPlace.A=0
Ponto_STR[Pallet_2,Prdt_15CoffeCrisp,7].OffsetPlace.B=0
Ponto_STR[Pallet_2,Prdt_15CoffeCrisp,7].OffsetPlace.C=0
;ENDFOLD
;ENDFOLD

;ENDFOLD
;FOLD LAYER 2: PLACE 8 ate 14
;FOLD PLACE 8
;FOLD PROPRIEDADES
Ponto_STR[Pallet_2,Prdt_15CoffeCrisp,8].NumCaixas = 1
Ponto_STR[Pallet_2,Prdt_15CoffeCrisp,8].PickOp = 6
Ponto_STR[Pallet_2,Prdt_15CoffeCrisp,8].ConfGarraOp = 5
Ponto_STR[Pallet_2,Prdt_15CoffeCrisp,8].FechaGarraOp = 0
Ponto_STR[Pallet_2,Prdt_15CoffeCrisp,8].AbreGarraOp = 0
Ponto_STR[Pallet_2,Prdt_15CoffeCrisp,8].SensoresCaixa = 1
Ponto_STR[Pallet_2,Prdt_15CoffeCrisp,8].TravaGarra = False
Ponto_STR[Pallet_2,Prdt_15CoffeCrisp,8].SkipGoHome = False
Ponto_STR[Pallet_2,Prdt_15CoffeCrisp,8].SkipSobeRelativo = False
Ponto_STR[Pallet_2,Prdt_15CoffeCrisp,8].XApp1Place=P2_15CoffeCrisp_8_App1
Ponto_STR[Pallet_2,Prdt_15CoffeCrisp,8].XApp2Place=P2_15CoffeCrisp_8_App2
Ponto_STR[Pallet_2,Prdt_15CoffeCrisp,8].XPlace=P2_15CoffeCrisp_8_Place
;ENDFOLD
;FOLD OffsetPlace
Ponto_STR[Pallet_2,Prdt_15CoffeCrisp,8].OffsetPlace.X=0
Ponto_STR[Pallet_2,Prdt_15CoffeCrisp,8].OffsetPlace.Y=0
Ponto_STR[Pallet_2,Prdt_15CoffeCrisp,8].OffsetPlace.Z=0
Ponto_STR[Pallet_2,Prdt_15CoffeCrisp,8].OffsetPlace.A=0
Ponto_STR[Pallet_2,Prdt_15CoffeCrisp,8].OffsetPlace.B=0
Ponto_STR[Pallet_2,Prdt_15CoffeCrisp,8].OffsetPlace.C=0
;ENDFOLD
;ENDFOLD

;FOLD PLACE 9
;FOLD PROPRIEDADES
Ponto_STR[Pallet_2,Prdt_15CoffeCrisp,9].NumCaixas = 1
Ponto_STR[Pallet_2,Prdt_15CoffeCrisp,9].PickOp = 6
Ponto_STR[Pallet_2,Prdt_15CoffeCrisp,9].ConfGarraOp = 5
Ponto_STR[Pallet_2,Prdt_15CoffeCrisp,9].FechaGarraOp = 0
Ponto_STR[Pallet_2,Prdt_15CoffeCrisp,9].AbreGarraOp = 0
Ponto_STR[Pallet_2,Prdt_15CoffeCrisp,9].SensoresCaixa = 1
Ponto_STR[Pallet_2,Prdt_15CoffeCrisp,9].TravaGarra = False
Ponto_STR[Pallet_2,Prdt_15CoffeCrisp,9].SkipGoHome = False
Ponto_STR[Pallet_2,Prdt_15CoffeCrisp,9].SkipSobeRelativo = False
Ponto_STR[Pallet_2,Prdt_15CoffeCrisp,9].XApp1Place=P2_15CoffeCrisp_9_App1
Ponto_STR[Pallet_2,Prdt_15CoffeCrisp,9].XApp2Place=P2_15CoffeCrisp_9_App2
Ponto_STR[Pallet_2,Prdt_15CoffeCrisp,9].XPlace=P2_15CoffeCrisp_9_Place
;ENDFOLD
;FOLD OffsetPlace
Ponto_STR[Pallet_2,Prdt_15CoffeCrisp,9].OffsetPlace.X=0
Ponto_STR[Pallet_2,Prdt_15CoffeCrisp,9].OffsetPlace.Y=0
Ponto_STR[Pallet_2,Prdt_15CoffeCrisp,9].OffsetPlace.Z=0
Ponto_STR[Pallet_2,Prdt_15CoffeCrisp,9].OffsetPlace.A=0
Ponto_STR[Pallet_2,Prdt_15CoffeCrisp,9].OffsetPlace.B=0
Ponto_STR[Pallet_2,Prdt_15CoffeCrisp,9].OffsetPlace.C=0
;ENDFOLD
;ENDFOLD

;FOLD PLACE 10
;FOLD PROPRIEDADES
Ponto_STR[Pallet_2,Prdt_15CoffeCrisp,10].NumCaixas = 1
Ponto_STR[Pallet_2,Prdt_15CoffeCrisp,10].PickOp = 6
Ponto_STR[Pallet_2,Prdt_15CoffeCrisp,10].ConfGarraOp = 5
Ponto_STR[Pallet_2,Prdt_15CoffeCrisp,10].FechaGarraOp = 0
Ponto_STR[Pallet_2,Prdt_15CoffeCrisp,10].AbreGarraOp = 0
Ponto_STR[Pallet_2,Prdt_15CoffeCrisp,10].SensoresCaixa = 1
Ponto_STR[Pallet_2,Prdt_15CoffeCrisp,10].TravaGarra = False
Ponto_STR[Pallet_2,Prdt_15CoffeCrisp,10].SkipGoHome = False
Ponto_STR[Pallet_2,Prdt_15CoffeCrisp,10].SkipSobeRelativo = False
Ponto_STR[Pallet_2,Prdt_15CoffeCrisp,10].XApp1Place=P2_15CoffeCrisp_10_App1
Ponto_STR[Pallet_2,Prdt_15CoffeCrisp,10].XApp2Place=P2_15CoffeCrisp_10_App2
Ponto_STR[Pallet_2,Prdt_15CoffeCrisp,10].XPlace=P2_15CoffeCrisp_10_Place
;ENDFOLD
;FOLD OffsetPlace
Ponto_STR[Pallet_2,Prdt_15CoffeCrisp,10].OffsetPlace.X=0
Ponto_STR[Pallet_2,Prdt_15CoffeCrisp,10].OffsetPlace.Y=0
Ponto_STR[Pallet_2,Prdt_15CoffeCrisp,10].OffsetPlace.Z=0
Ponto_STR[Pallet_2,Prdt_15CoffeCrisp,10].OffsetPlace.A=0
Ponto_STR[Pallet_2,Prdt_15CoffeCrisp,10].OffsetPlace.B=0
Ponto_STR[Pallet_2,Prdt_15CoffeCrisp,10].OffsetPlace.C=0
;ENDFOLD
;ENDFOLD

;FOLD PLACE 11
;FOLD PROPRIEDADES
Ponto_STR[Pallet_2,Prdt_15CoffeCrisp,11].NumCaixas = 2
Ponto_STR[Pallet_2,Prdt_15CoffeCrisp,11].PickOp = 8
Ponto_STR[Pallet_2,Prdt_15CoffeCrisp,11].ConfGarraOp = 5
Ponto_STR[Pallet_2,Prdt_15CoffeCrisp,11].FechaGarraOp = 0
Ponto_STR[Pallet_2,Prdt_15CoffeCrisp,11].AbreGarraOp = 1
Ponto_STR[Pallet_2,Prdt_15CoffeCrisp,11].SensoresCaixa = 123
Ponto_STR[Pallet_2,Prdt_15CoffeCrisp,11].TravaGarra = True
Ponto_STR[Pallet_2,Prdt_15CoffeCrisp,11].SkipGoHome = False
Ponto_STR[Pallet_2,Prdt_15CoffeCrisp,11].SkipSobeRelativo = False
Ponto_STR[Pallet_2,Prdt_15CoffeCrisp,11].XApp1Place=P2_15CoffeCrisp_11_App1
Ponto_STR[Pallet_2,Prdt_15CoffeCrisp,11].XApp2Place=P2_15CoffeCrisp_11_App2
Ponto_STR[Pallet_2,Prdt_15CoffeCrisp,11].XPlace=P2_15CoffeCrisp_11_Place
;ENDFOLD
;FOLD OffsetPlace
Ponto_STR[Pallet_2,Prdt_15CoffeCrisp,11].OffsetPlace.X=0
Ponto_STR[Pallet_2,Prdt_15CoffeCrisp,11].OffsetPlace.Y=0
Ponto_STR[Pallet_2,Prdt_15CoffeCrisp,11].OffsetPlace.Z=0
Ponto_STR[Pallet_2,Prdt_15CoffeCrisp,11].OffsetPlace.A=0
Ponto_STR[Pallet_2,Prdt_15CoffeCrisp,11].OffsetPlace.B=0
Ponto_STR[Pallet_2,Prdt_15CoffeCrisp,11].OffsetPlace.C=0
;ENDFOLD
;ENDFOLD

;FOLD PLACE 12
;FOLD PROPRIEDADES
Ponto_STR[Pallet_2,Prdt_15CoffeCrisp,12].NumCaixas = 2
Ponto_STR[Pallet_2,Prdt_15CoffeCrisp,12].PickOp = 8
Ponto_STR[Pallet_2,Prdt_15CoffeCrisp,12].ConfGarraOp = 5
Ponto_STR[Pallet_2,Prdt_15CoffeCrisp,12].FechaGarraOp = 0
Ponto_STR[Pallet_2,Prdt_15CoffeCrisp,12].AbreGarraOp = 1
Ponto_STR[Pallet_2,Prdt_15CoffeCrisp,12].SensoresCaixa = 123
Ponto_STR[Pallet_2,Prdt_15CoffeCrisp,12].TravaGarra = True
Ponto_STR[Pallet_2,Prdt_15CoffeCrisp,12].SkipGoHome = False
Ponto_STR[Pallet_2,Prdt_15CoffeCrisp,12].SkipSobeRelativo = False
Ponto_STR[Pallet_2,Prdt_15CoffeCrisp,12].XApp1Place=P2_15CoffeCrisp_12_App1
Ponto_STR[Pallet_2,Prdt_15CoffeCrisp,12].XApp2Place=P2_15CoffeCrisp_12_App2
Ponto_STR[Pallet_2,Prdt_15CoffeCrisp,12].XPlace=P2_15CoffeCrisp_12_Place
;ENDFOLD
;FOLD OffsetPlace
Ponto_STR[Pallet_2,Prdt_15CoffeCrisp,12].OffsetPlace.X=0
Ponto_STR[Pallet_2,Prdt_15CoffeCrisp,12].OffsetPlace.Y=0
Ponto_STR[Pallet_2,Prdt_15CoffeCrisp,12].OffsetPlace.Z=0
Ponto_STR[Pallet_2,Prdt_15CoffeCrisp,12].OffsetPlace.A=0
Ponto_STR[Pallet_2,Prdt_15CoffeCrisp,12].OffsetPlace.B=0
Ponto_STR[Pallet_2,Prdt_15CoffeCrisp,12].OffsetPlace.C=0
;ENDFOLD
;ENDFOLD

;FOLD PLACE 13
;FOLD PROPRIEDADES
Ponto_STR[Pallet_2,Prdt_15CoffeCrisp,13].NumCaixas = 3
Ponto_STR[Pallet_2,Prdt_15CoffeCrisp,13].PickOp = 6
Ponto_STR[Pallet_2,Prdt_15CoffeCrisp,13].ConfGarraOp = 5
Ponto_STR[Pallet_2,Prdt_15CoffeCrisp,13].FechaGarraOp = 0
Ponto_STR[Pallet_2,Prdt_15CoffeCrisp,13].AbreGarraOp = 1
Ponto_STR[Pallet_2,Prdt_15CoffeCrisp,13].SensoresCaixa = 1234
Ponto_STR[Pallet_2,Prdt_15CoffeCrisp,13].TravaGarra = True
Ponto_STR[Pallet_2,Prdt_15CoffeCrisp,13].SkipGoHome = False
Ponto_STR[Pallet_2,Prdt_15CoffeCrisp,13].SkipSobeRelativo = False
Ponto_STR[Pallet_2,Prdt_15CoffeCrisp,13].XApp1Place=P2_15CoffeCrisp_13_App1
Ponto_STR[Pallet_2,Prdt_15CoffeCrisp,13].XApp2Place=P2_15CoffeCrisp_13_App2
Ponto_STR[Pallet_2,Prdt_15CoffeCrisp,13].XPlace=P2_15CoffeCrisp_13_Place
;ENDFOLD
;FOLD OffsetPlace
Ponto_STR[Pallet_2,Prdt_15CoffeCrisp,13].OffsetPlace.X=0
Ponto_STR[Pallet_2,Prdt_15CoffeCrisp,13].OffsetPlace.Y=0
Ponto_STR[Pallet_2,Prdt_15CoffeCrisp,13].OffsetPlace.Z=0
Ponto_STR[Pallet_2,Prdt_15CoffeCrisp,13].OffsetPlace.A=0
Ponto_STR[Pallet_2,Prdt_15CoffeCrisp,13].OffsetPlace.B=0
Ponto_STR[Pallet_2,Prdt_15CoffeCrisp,13].OffsetPlace.C=0
;ENDFOLD
;ENDFOLD

;FOLD PLACE 14
;FOLD PROPRIEDADES
Ponto_STR[Pallet_2,Prdt_15CoffeCrisp,14].NumCaixas = 3
Ponto_STR[Pallet_2,Prdt_15CoffeCrisp,14].PickOp = 6
Ponto_STR[Pallet_2,Prdt_15CoffeCrisp,14].ConfGarraOp = 5
Ponto_STR[Pallet_2,Prdt_15CoffeCrisp,14].FechaGarraOp = 0
Ponto_STR[Pallet_2,Prdt_15CoffeCrisp,14].AbreGarraOp = 1
Ponto_STR[Pallet_2,Prdt_15CoffeCrisp,14].SensoresCaixa = 1234
Ponto_STR[Pallet_2,Prdt_15CoffeCrisp,14].TravaGarra = True
Ponto_STR[Pallet_2,Prdt_15CoffeCrisp,14].SkipGoHome = False
Ponto_STR[Pallet_2,Prdt_15CoffeCrisp,14].SkipSobeRelativo = False
Ponto_STR[Pallet_2,Prdt_15CoffeCrisp,14].XApp1Place=P2_15CoffeCrisp_14_App1
Ponto_STR[Pallet_2,Prdt_15CoffeCrisp,14].XApp2Place=P2_15CoffeCrisp_14_App2
Ponto_STR[Pallet_2,Prdt_15CoffeCrisp,14].XPlace=P2_15CoffeCrisp_14_Place
;ENDFOLD
;FOLD OffsetPlace
Ponto_STR[Pallet_2,Prdt_15CoffeCrisp,14].OffsetPlace.X=0
Ponto_STR[Pallet_2,Prdt_15CoffeCrisp,14].OffsetPlace.Y=0
Ponto_STR[Pallet_2,Prdt_15CoffeCrisp,14].OffsetPlace.Z=0
Ponto_STR[Pallet_2,Prdt_15CoffeCrisp,14].OffsetPlace.A=0
Ponto_STR[Pallet_2,Prdt_15CoffeCrisp,14].OffsetPlace.B=0
Ponto_STR[Pallet_2,Prdt_15CoffeCrisp,14].OffsetPlace.C=0
;ENDFOLD
;ENDFOLD

;ENDFOLD
;ENDFOLD

;ENDFOLD
END

--- TMatriz.dat ---
&ACCESS RV1
DEFDAT Ponto_STR_Iniciar PUBLIC
;FOLD PALLET 1
;FOLD Pallet 1 - Produto 9Aero
;FOLD PLACE 1
DECL E6POS P1_9Aero_1_App1={X 1022.73301,Y -522.76885,Z 1064.59491,A 180,B 0,C -180,S 2,T 2,E1 0,E2 0,E3 0,E4 0,E5 0,E6 0}
DECL E6POS P1_9Aero_1_App2={X 1022.73295,Y -522.7684,Z 964.59495,A 180,B 0,C 180,S 2,T 2,E1 0,E2 0,E3 0,E4 0,E5 0,E6 0}
DECL E6POS P1_9Aero_1_Place={X 1122.73281,Y -522.76864,Z 814.59517,A -180,B 0,C -180,S 2,T 2,E1 0,E2 0,E3 0,E4 0,E5 0,E6 0}
;ENDFOLD

;FOLD PLACE 2
DECL E6POS P1_9Aero_2_App1={X 536.73295,Y -522.76875,Z 1064.59497,A 180,B 0,C 180,S 2,T 2,E1 0,E2 0,E3 0,E4 0,E5 0,E6 0}
DECL E6POS P1_9Aero_2_App2={X 536.73295,Y -522.76869,Z 964.59466,A -180,B 0,C -180,S 2,T 2,E1 0,E2 0,E3 0,E4 0,E5 0,E6 0}
DECL E6POS P1_9Aero_2_Place={X 586.73291,Y -522.76888,Z 814.59521,A 180,B 0,C -180,S 2,T 2,E1 0,E2 0,E3 0,E4 0,E5 0,E6 0}
;ENDFOLD

;ENDFOLD

;FOLD Pallet 1 - Produto 5Aero
;FOLD PLACE 1
DECL E6POS P1_5Aero_1_App1={X 1100.19092,Y -381.19586,Z 1064.5593,A -180,B 0,C -180,S 2,T 2,E1 0,E2 0,E3 0,E4 0,E5 0,E6 0}
DECL E6POS P1_5Aero_1_App2={X 1100.19089,Y -381.19558,Z 914.55891,A -180,B 0,C -180,S 2,T 2,E1 0,E2 0,E3 0,E4 0,E5 0,E6 0}
DECL E6POS P1_5Aero_1_Place={X 1200.19026,Y -381.19557,Z 814.55914,A 180,B 0,C 180,S 2,T 2,E1 0,E2 0,E3 0,E4 0,E5 0,E6 0}
;ENDFOLD

;FOLD PLACE 2
DECL E6POS P1_5Aero_2_App1={X 740.19091,Y -381.19584,Z 1064.55897,A 180,B 0,C -180,S 2,T 2,E1 0,E2 0,E3 0,E4 0,E5 0,E6 0}
DECL E6POS P1_5Aero_2_App2={X 740.19091,Y -381.19576,Z 914.55853,A 180,B 0,C -180,S 2,T 2,E1 0,E2 0,E3 0,E4 0,E5 0,E6 0}
DECL E6POS P1_5Aero_2_Place={X 840.19068,Y -381.19567,Z 814.55885,A 180,B 0,C 180,S 2,T 2,E1 0,E2 0,E3 0,E4 0,E5 0,E6 0}
;ENDFOLD

;FOLD PLACE 3
DECL E6POS P1_5Aero_3_App1={X 380.19048,Y -381.19555,Z 1064.55905,A -180,B 0,C -180,S 2,T 2,E1 0,E2 0,E3 0,E4 0,E5 0,E6 0}
DECL E6POS P1_5Aero_3_App2={X 380.1905,Y -381.19547,Z 914.5591,A -180,B 0,C 180,S 2,T 2,E1 0,E2 0,E3 0,E4 0,E5 0,E6 0}
DECL E6POS P1_5Aero_3_Place={X 480.1904,Y -381.19581,Z 814.55931,A -180,B 0,C -180,S 2,T 2,E1 0,E2 0,E3 0,E4 0,E5 0,E6 0}
;ENDFOLD

;ENDFOLD

;FOLD Pallet 1 - Produto 2Aero
;FOLD PLACE 1
DECL E6POS P1_2Aero_1_App1={X 656.91511,Y -930.82109,Z 1114.55821,A 90,B 0,C -180,S 2,T 2,E1 0,E2 0,E3 0,E4 0,E5 0,E6 0}
DECL E6POS P1_2Aero_1_App2={X 656.91452,Y -930.82084,Z 914.55794,A 90,B 0,C -180,S 2,T 2,E1 0,E2 0,E3 0,E4 0,E5 0,E6 0}
DECL E6POS P1_2Aero_1_Place={X 656.91466,Y -1030.82103,Z 814.55883,A 90,B 0,C -180,S 2,T 2,E1 0,E2 0,E3 0,E4 0,E5 0,E6 0}
;ENDFOLD

;FOLD PLACE 2
DECL E6POS P1_2Aero_2_App1={X 656.91475,Y -619.82119,Z 1114.55821,A 90,B 0,C -180,S 2,T 2,E1 0,E2 0,E3 0,E4 0,E5 0,E6 0}
DECL E6POS P1_2Aero_2_App2={X 656.9148,Y -619.82082,Z 914.55773,A 90,B 0,C -180,S 2,T 2,E1 0,E2 0,E3 0,E4 0,E5 0,E6 0}
DECL E6POS P1_2Aero_2_Place={X 656.91513,Y -719.82119,Z 814.55847,A 90,B 0,C -180,S 2,T 2,E1 0,E2 0,E3 0,E4 0,E5 0,E6 0}
;ENDFOLD

;FOLD PLACE 3
DECL E6POS P1_2Aero_3_App1={X 656.91433,Y -308.82121,Z 1114.55796,A 90,B 0,C -180,S 2,T 2,E1 0,E2 0,E3 0,E4 0,E5 0,E6 0}
DECL E6POS P1_2Aero_3_App2={X 656.9144,Y -308.82081,Z 914.55753,A 90,B 0,C -180,S 2,T 2,E1 0,E2 0,E3 0,E4 0,E5 0,E6 0}
DECL E6POS P1_2Aero_3_Place={X 656.9151,Y -408.82095,Z 814.55837,A 90,B 0,C -180,S 2,T 2,E1 0,E2 0,E3 0,E4 0,E5 0,E6 0}
;ENDFOLD

;ENDFOLD

;FOLD Pallet 1 - Produto 11CoffeCrisp
;FOLD PLACE 1
DECL E6POS P1_11CoffeCrisp_1_App1={X 1151.36818,Y -373.97179,Z 1064.54984,A 180,B 0,C -180,S 2,T 2,E1 0,E2 0,E3 0,E4 0,E5 0,E6 0}
DECL E6POS P1_11CoffeCrisp_1_App2={X 1151.36819,Y -373.97194,Z 964.54979,A 180,B 0,C -180,S 2,T 2,E1 0,E2 0,E3 0,E4 0,E5 0,E6 0}
DECL E6POS P1_11CoffeCrisp_1_Place={X 1251.36773,Y -373.97178,Z 814.55016,A 180,B 0,C -180,S 2,T 2,E1 0,E2 0,E3 0,E4 0,E5 0,E6 0}
;ENDFOLD

;FOLD PLACE 2
DECL E6POS P1_11CoffeCrisp_2_App1={X 757.36709,Y -373.97196,Z 1064.55048,A 180,B 0,C -180,S 2,T 2,E1 0,E2 0,E3 0,E4 0,E5 0,E6 0}
DECL E6POS P1_11CoffeCrisp_2_App2={X 757.36707,Y -373.97216,Z 964.55002,A 180,B 0,C 180,S 2,T 2,E1 0,E2 0,E3 0,E4 0,E5 0,E6 0}
DECL E6POS P1_11CoffeCrisp_2_Place={X 857.36783,Y -373.97166,Z 814.55037,A 180,B 0,C -180,S 2,T 2,E1 0,E2 0,E3 0,E4 0,E5 0,E6 0}
;ENDFOLD

;FOLD PLACE 3
DECL E6POS P1_11CoffeCrisp_3_App1={X 363.36776,Y -373.97205,Z 1064.54992,A 180,B 0,C -180,S 2,T 2,E1 0,E2 0,E3 0,E4 0,E5 0,E6 0}
DECL E6POS P1_11CoffeCrisp_3_App2={X 363.36773,Y -373.97215,Z 964.55039,A 180,B 0,C -180,S 2,T 2,E1 0,E2 0,E3 0,E4 0,E5 0,E6 0}
DECL E6POS P1_11CoffeCrisp_3_Place={X 463.36751,Y -373.97168,Z 814.54997,A 180,B 0,C 180,S 2,T 2,E1 0,E2 0,E3 0,E4 0,E5 0,E6 0}
;ENDFOLD

;ENDFOLD

;FOLD Pallet 1 - Produto 17KitKat
;FOLD PLACE 1
DECL E6POS P1_17KitKat_1_App1={X 1164.97122,Y -349.70187,Z 1114.5871,A 180,B 0,C -180,S 2,T 2,E1 0,E2 0,E3 0,E4 0,E5 0,E6 0}
DECL E6POS P1_17KitKat_1_App2={X 1164.97124,Y -349.70201,Z 964.58697,A 180,B 0,C 180,S 2,T 2,E1 0,E2 0,E3 0,E4 0,E5 0,E6 0}
DECL E6POS P1_17KitKat_1_Place={X 1264.97156,Y -349.7018,Z 814.58693,A 180,B 0,C -180,S 2,T 2,E1 0,E2 0,E3 0,E4 0,E5 0,E6 0}
;ENDFOLD

;FOLD PLACE 2
DECL E6POS P1_17KitKat_2_App1={X 864.97244,Y -349.70175,Z 1114.58691,A 180,B 0,C 180,S 2,T 2,E1 0,E2 0,E3 0,E4 0,E5 0,E6 0}
DECL E6POS P1_17KitKat_2_App2={X 864.97244,Y -349.70212,Z 964.58694,A 180,B 0,C -180,S 2,T 2,E1 0,E2 0,E3 0,E4 0,E5 0,E6 0}
DECL E6POS P1_17KitKat_2_Place={X 964.97194,Y -349.70202,Z 814.58663,A 180,B 0,C 180,S 2,T 2,E1 0,E2 0,E3 0,E4 0,E5 0,E6 0}
;ENDFOLD

;FOLD PLACE 3
DECL E6POS P1_17KitKat_3_App1={X 564.97231,Y -349.70207,Z 1114.58678,A -180,B 0,C 180,S 2,T 2,E1 0,E2 0,E3 0,E4 0,E5 0,E6 0}
DECL E6POS P1_17KitKat_3_App2={X 564.97232,Y -349.70204,Z 964.58683,A -180,B 0,C -180,S 2,T 2,E1 0,E2 0,E3 0,E4 0,E5 0,E6 0}
DECL E6POS P1_17KitKat_3_Place={X 664.97218,Y -349.70207,Z 814.5867,A 180,B 0,C -180,S 2,T 2,E1 0,E2 0,E3 0,E4 0,E5 0,E6 0}
;ENDFOLD

;FOLD PLACE 4
DECL E6POS P1_17KitKat_4_App1={X 314.97216,Y -349.70215,Z 1114.58736,A -180,B 0,C -180,S 2,T 2,E1 0,E2 0,E3 0,E4 0,E5 0,E6 0}
DECL E6POS P1_17KitKat_4_App2={X 314.97221,Y -349.702,Z 964.5866,A 180,B 0,C -180,S 2,T 2,E1 0,E2 0,E3 0,E4 0,E5 0,E6 0}
DECL E6POS P1_17KitKat_4_Place={X 364.97196,Y -349.70185,Z 814.58667,A -180,B 0,C 180,S 2,T 2,E1 0,E2 0,E3 0,E4 0,E5 0,E6 0}
;ENDFOLD

;ENDFOLD

;FOLD Pallet 1 - Produto 19KitKat
;FOLD PLACE 1
DECL E6POS P1_19KitKat_1_App1={X 627.17081,Y -1004.18327,Z 964.60036,A 90,B 0,C 180,S 2,T 2,E1 0,E2 0,E3 0,E4 0,E5 0,E6 0}
DECL E6POS P1_19KitKat_1_App2={X 627.17081,Y -1004.18312,Z 914.60037,A 90,B 0,C -180,S 2,T 2,E1 0,E2 0,E3 0,E4 0,E5 0,E6 0}
DECL E6POS P1_19KitKat_1_Place={X 627.17081,Y -1054.18351,Z 814.59956,A 90,B 0,C -180,S 2,T 2,E1 0,E2 0,E3 0,E4 0,E5 0,E6 0}
;ENDFOLD

;FOLD PLACE 2
DECL E6POS P1_19KitKat_2_App1={X 627.17081,Y -663.1828,Z 964.59988,A 90,B 0,C -180,S 2,T 2,E1 0,E2 0,E3 0,E4 0,E5 0,E6 0}
DECL E6POS P1_19KitKat_2_App2={X 627.17081,Y -663.18258,Z 914.60023,A 90,B 0,C -180,S 2,T 2,E1 0,E2 0,E3 0,E4 0,E5 0,E6 0}
DECL E6POS P1_19KitKat_2_Place={X 627.16999,Y -713.18307,Z 814.59982,A 90,B 0,C -180,S 2,T 2,E1 0,E2 0,E3 0,E4 0,E5 0,E6 0}
;ENDFOLD

;FOLD PLACE 3
DECL E6POS P1_19KitKat_3_App1={X 627.17081,Y -322.18314,Z 964.60008,A 90,B 0,C 180,S 2,T 2,E1 0,E2 0,E3 0,E4 0,E5 0,E6 0}
DECL E6POS P1_19KitKat_3_App2={X 627.17081,Y -322.18283,Z 914.59997,A 90,B 0,C -180,S 2,T 2,E1 0,E2 0,E3 0,E4 0,E5 0,E6 0}
DECL E6POS P1_19KitKat_3_Place={X 627.17051,Y -372.18279,Z 814.59944,A 90,B 0,C 180,S 2,T 2,E1 0,E2 0,E3 0,E4 0,E5 0,E6 0}
;ENDFOLD

;FOLD PLACE 4
DECL E6POS P1_19KitKat_4_App1={X 934.59434,Y -397.19007,Z 964.60022,A 180,B 0,C -180,S 2,T 2,E1 0,E2 0,E3 0,E4 0,E5 0,E6 0}
DECL E6POS P1_19KitKat_4_App2={X 934.59395,Y -397.18983,Z 914.60038,A -180,B 0,C -180,S 2,T 2,E1 0,E2 0,E3 0,E4 0,E5 0,E6 0}
DECL E6POS P1_19KitKat_4_Place={X 984.59395,Y -397.18983,Z 814.60016,A 180,B 0,C -180,S 2,T 2,E1 0,E2 0,E3 0,E4 0,E5 0,E6 0}
;ENDFOLD

;FOLD PLACE 5
DECL E6POS P1_19KitKat_5_App1={X 636.59337,Y -397.19032,Z 964.59991,A 180,B 0,C -180,S 2,T 2,E1 0,E2 0,E3 0,E4 0,E5 0,E6 0}
DECL E6POS P1_19KitKat_5_App2={X 636.59358,Y -397.19003,Z 914.59977,A -180,B 0,C -180,S 2,T 2,E1 0,E2 0,E3 0,E4 0,E5 0,E6 0}
DECL E6POS P1_19KitKat_5_Place={X 686.59358,Y -397.19003,Z 814.60016,A -180,B 0,C 180,S 2,T 2,E1 0,E2 0,E3 0,E4 0,E5 0,E6 0}
;ENDFOLD

;FOLD PLACE 6
DECL E6POS P1_19KitKat_6_App1={X 338.58782,Y -397.19008,Z 964.59943,A -180,B 0,C -180,S 2,T 2,E1 0,E2 0,E3 0,E4 0,E5 0,E6 0}
DECL E6POS P1_19KitKat_6_App2={X 338.58782,Y -397.19003,Z 914.60003,A -180,B 0,C 180,S 2,T 2,E1 0,E2 0,E3 0,E4 0,E5 0,E6 0}
DECL E6POS P1_19KitKat_6_Place={X 388.58782,Y -397.19974,Z 814.59632,A -180,B 0,C 180,S 2,T 2,E1 0,E2 0,E3 0,E4 0,E5 0,E6 0}
;ENDFOLD

;FOLD PLACE 7
DECL E6POS P1_19KitKat_7_App1={X 627.79688,Y -1005.14358,Z 970.012,A 90,B 0,C 180,S 2,T 2,E1 0,E2 0,E3 0,E4 0,E5 0,E6 0}
DECL E6POS P1_19KitKat_7_App2={X 627.79716,Y -1005.14347,Z 900.012,A 90,B 0,C -180,S 2,T 2,E1 0,E2 0,E3 0,E4 0,E5 0,E6 0}
DECL E6POS P1_19KitKat_7_Place={X 627.79716,Y -1055.14347,Z 814.611,A 90,B 0,C -180,S 2,T 2,E1 0,E2 0,E3 0,E4 0,E5 0,E6 0}
;ENDFOLD

;FOLD PLACE 8
DECL E6POS P1_19KitKat_8_App1={X 627.79702,Y -664.19505,Z 970.012,A 90,B 0,C -180,S 2,T 2,E1 0,E2 0,E3 0,E4 0,E5 0,E6 0}
DECL E6POS P1_19KitKat_8_App2={X 627.79702,Y -664.19491,Z 900.012,A 90,B 0,C -180,S 2,T 2,E1 0,E2 0,E3 0,E4 0,E5 0,E6 0}
DECL E6POS P1_19KitKat_8_Place={X 627.79674,Y -714.19509,Z 814.587,A 90,B 0,C 180,S 2,T 2,E1 0,E2 0,E3 0,E4 0,E5 0,E6 0}
;ENDFOLD

;FOLD PLACE 9
DECL E6POS P1_19KitKat_9_App1={X 627.79265,Y -323.14959,Z 970.012,A 90,B 0,C -180,S 2,T 2,E1 0,E2 0,E3 0,E4 0,E5 0,E6 0}
DECL E6POS P1_19KitKat_9_App2={X 627.79262,Y -323.14974,Z 900.012,A 90,B 0,C -180,S 2,T 2,E1 0,E2 0,E3 0,E4 0,E5 0,E6 0}
DECL E6POS P1_19KitKat_9_Place={X 627.79299,Y -373.1496,Z 814.595,A 90,B 0,C -180,S 2,T 2,E1 0,E2 0,E3 0,E4 0,E5 0,E6 0}
;ENDFOLD

;FOLD PLACE 10
DECL E6POS P1_19KitKat_10_App1={X 683.56502,Y -397.17408,Z 970.012,A -180,B 0,C 180,S 2,T 2,E1 0,E2 0,E3 0,E4 0,E5 0,E6 0}
DECL E6POS P1_19KitKat_10_App2={X 683.56511,Y -397.17413,Z 899.8,A -180,B 0,C -180,S 2,T 2,E1 0,E2 0,E3 0,E4 0,E5 0,E6 0}
DECL E6POS P1_19KitKat_10_Place={X 633.56511,Y -397.17413,Z 814.617,A 180,B 0,C 180,S 2,T 2,E1 0,E2 0,E3 0,E4 0,E5 0,E6 0}
;ENDFOLD

;FOLD PLACE 11
DECL E6POS P1_19KitKat_11_App1={X 981.57268,Y -397.18858,Z 970.012,A -180,B 0,C -180,S 2,T 2,E1 0,E2 0,E3 0,E4 0,E5 0,E6 0}
DECL E6POS P1_19KitKat_11_App2={X 981.57236,Y -397.18838,Z 899.8,A -180,B 0,C -180,S 2,T 2,E1 0,E2 0,E3 0,E4 0,E5 0,E6 0}
DECL E6POS P1_19KitKat_11_Place={X 931.57236,Y -397.18838,Z 814.603,A -180,B 0,C -180,S 2,T 2,E1 0,E2 0,E3 0,E4 0,E5 0,E6 0}
;ENDFOLD

;FOLD PLACE 12
DECL E6POS P1_19KitKat_12_App1={X 1269.56898,Y -397.18832,Z 970.012,A 180,B 0,C -180,S 2,T 2,E1 0,E2 0,E3 0,E4 0,E5 0,E6 0}
DECL E6POS P1_19KitKat_12_App2={X 1269.56898,Y -397.18838,Z 899.8,A -180,B 0,C -180,S 2,T 2,E1 0,E2 0,E3 0,E4 0,E5 0,E6 0}
DECL E6POS P1_19KitKat_12_Place={X 1229.56898,Y -397.18174,Z 814.61,A -180,B 0,C -180,S 2,T 2,E1 0,E2 0,E3 0,E4 0,E5 0,E6 0}
;ENDFOLD

;ENDFOLD

;FOLD Pallet 1 - Produto 20KitKat
;FOLD PLACE 1
DECL E6POS P1_20KitKat_1_App1={X 632.10189,Y -938.77405,Z 984.5769,A 90,B 0,C 180,S 2,T 2,E1 0,E2 0,E3 0,E4 0,E5 0,E6 0}
DECL E6POS P1_20KitKat_1_App2={X 632.10188,Y -938.77417,Z 864.57961,A 90,B 0,C -180,S 2,T 2,E1 0,E2 0,E3 0,E4 0,E5 0,E6 0}
DECL E6POS P1_20KitKat_1_Place={X 632.10155,Y -1038.77384,Z 814.57747,A 90,B 0,C -180,S 2,T 2,E1 0,E2 0,E3 0,E4 0,E5 0,E6 0}
;ENDFOLD

;FOLD PLACE 2
DECL E6POS P1_20KitKat_2_App1={X 632.08454,Y -672.77189,Z 984.57621,A 90,B 0,C 180,S 2,T 2,E1 0,E2 0,E3 0,E4 0,E5 0,E6 0}
DECL E6POS P1_20KitKat_2_App2={X 632.08454,Y -672.7719,Z 864.57961,A 90,B 0,C 180,S 2,T 2,E1 0,E2 0,E3 0,E4 0,E5 0,E6 0}
DECL E6POS P1_20KitKat_2_Place={X 632.08454,Y -722.7719,Z 814.57773,A 90,B 0,C 180,S 2,T 2,E1 0,E2 0,E3 0,E4 0,E5 0,E6 0}
;ENDFOLD

;FOLD PLACE 3
DECL E6POS P1_20KitKat_3_App1={X 632.10156,Y -356.7796,Z 984.57723,A 90,B 0,C -180,S 2,T 2,E1 0,E2 0,E3 0,E4 0,E5 0,E6 0}
DECL E6POS P1_20KitKat_3_App2={X 632.10172,Y -356.7796,Z 864.57961,A 90,B 0,C 180,S 2,T 2,E1 0,E2 0,E3 0,E4 0,E5 0,E6 0}
DECL E6POS P1_20KitKat_3_Place={X 632.10155,Y -406.7796,Z 814.57711,A 90,B 0,C -180,S 2,T 2,E1 0,E2 0,E3 0,E4 0,E5 0,E6 0}
;ENDFOLD

;ENDFOLD

;FOLD Pallet 1 - Produto 21KitKat
;FOLD PLACE 1
DECL E6POS P1_21KitKat_1_App1={X 661.81794,Y -933.26894,Z 1064.51376,A 90,B 0,C -180,S 2,T 2,E1 0,E2 0,E3 0,E4 0,E5 0,E6 0}
DECL E6POS P1_21KitKat_1_App2={X 661.81796,Y -933.26883,Z 964.51401,A 90,B 0,C -180,S 2,T 2,E1 0,E2 0,E3 0,E4 0,E5 0,E6 0}
DECL E6POS P1_21KitKat_1_Place={X 661.81808,Y -1033.26888,Z 814.51394,A 90,B 0,C -180,S 2,T 2,E1 0,E2 0,E3 0,E4 0,E5 0,E6 0}
;ENDFOLD

;FOLD PLACE 2
DECL E6POS P1_21KitKat_2_App1={X 661.81739,Y -623.26907,Z 1064.51434,A 90,B 0,C -180,S 2,T 2,E1 0,E2 0,E3 0,E4 0,E5 0,E6 0}
DECL E6POS P1_21KitKat_2_App2={X 661.81738,Y -623.26912,Z 964.51429,A 90,B 0,C 180,S 2,T 2,E1 0,E2 0,E3 0,E4 0,E5 0,E6 0}
DECL E6POS P1_21KitKat_2_Place={X 661.8182,Y -723.26873,Z 814.51377,A 90,B 0,C -180,S 2,T 2,E1 0,E2 0,E3 0,E4 0,E5 0,E6 0}
;ENDFOLD

;FOLD PLACE 3
DECL E6POS P1_21KitKat_3_App1={X 661.81772,Y -313.26888,Z 1064.51417,A 90,B 0,C -180,S 2,T 2,E1 0,E2 0,E3 0,E4 0,E5 0,E6 0}
DECL E6POS P1_21KitKat_3_App2={X 661.81766,Y -313.26922,Z 964.51392,A 90,B 0,C 180,S 2,T 2,E1 0,E2 0,E3 0,E4 0,E5 0,E6 0}
DECL E6POS P1_21KitKat_3_Place={X 661.81803,Y -413.26929,Z 814.5136,A 90,B 0,C -180,S 2,T 2,E1 0,E2 0,E3 0,E4 0,E5 0,E6 0}
;ENDFOLD

;ENDFOLD

;FOLD Pallet 1 - Produto 23Smarties
;FOLD PLACE 1
DECL E6POS P1_23Smarties_1_App1={X 670.70243,Y -952.53077,Z 1158.21812,A 90,B 0,C -180,S 2,T 2,E1 0,E2 0,E3 0,E4 0,E5 0,E6 0}
DECL E6POS P1_23Smarties_1_App2={X 670.70243,Y -952.5308,Z 958.21659,A 90,B 0,C 180,S 2,T 2,E1 0,E2 0,E3 0,E4 0,E5 0,E6 0}
DECL E6POS P1_23Smarties_1_Place={X 720.70181,Y -1002.53052,Z 858.21764,A 90,B 0,C -180,S 2,T 2,E1 0,E2 0,E3 0,E4 0,E5 0,E6 0}
;ENDFOLD

;FOLD PLACE 2
DECL E6POS P1_23Smarties_2_App1={X 200.73141,Y -953.526,Z 1163.74438,A 90,B 0,C 180,S 2,T 2,E1 0,E2 0,E3 0,E4 0,E5 0,E6 0}
DECL E6POS P1_23Smarties_2_App2={X 200.731,Y -953.526,Z 958.21839,A 90,B 0,C -180,S 2,T 2,E1 0,E2 0,E3 0,E4 0,E5 0,E6 0}
DECL E6POS P1_23Smarties_2_Place={X 250.73131,Y -1003.52661,Z 858.21782,A 90,B 0,C -180,S 2,T 2,E1 0,E2 0,E3 0,E4 0,E5 0,E6 0}
;ENDFOLD

;FOLD PLACE 3
DECL E6POS P1_23Smarties_3_App1={X 670.70283,Y -448.53129,Z 1158.21841,A 90,B 0,C -180,S 2,T 2,E1 0,E2 0,E3 0,E4 0,E5 0,E6 0}
DECL E6POS P1_23Smarties_3_App2={X 670.70285,Y -448.53117,Z 958.21705,A 90,B 0,C -180,S 2,T 2,E1 0,E2 0,E3 0,E4 0,E5 0,E6 0}
DECL E6POS P1_23Smarties_3_Place={X 720.702,Y -498.53111,Z 858.21709,A 90,B 0,C -180,S 2,T 2,E1 0,E2 0,E3 0,E4 0,E5 0,E6 0}
;ENDFOLD

;FOLD PLACE 4
DECL E6POS P1_23Smarties_4_App1={X 200.73073,Y -449.52568,Z 1140.51235,A 90,B 0,C -180,S 2,T 2,E1 0,E2 0,E3 0,E4 0,E5 0,E6 0}
DECL E6POS P1_23Smarties_4_App2={X 200.7307,Y -449.52562,Z 958.21846,A 90,B 0,C -180,S 2,T 2,E1 0,E2 0,E3 0,E4 0,E5 0,E6 0}
DECL E6POS P1_23Smarties_4_Place={X 250.73049,Y -499.52567,Z 858.21817,A 90,B 0,C -180,S 2,T 2,E1 0,E2 0,E3 0,E4 0,E5 0,E6 0}
;ENDFOLD

;FOLD PLACE 5
DECL E6POS P1_23Smarties_5_App1={X 552.18218,Y -949.33572,Z 1158.22,A 90,B 0,C -180,S 2,T 2,E1 0,E2 0,E3 0,E4 0,E5 0,E6 0}
DECL E6POS P1_23Smarties_5_App2={X 552.18236,Y -949.33572,Z 958.217,A 90,B 0,C 180,S 2,T 2,E1 0,E2 0,E3 0,E4 0,E5 0,E6 0}
DECL E6POS P1_23Smarties_5_Place={X 502.18236,Y -999.33572,Z 858.218,A 90,B 0,C -180,S 2,T 2,E1 0,E2 0,E3 0,E4 0,E5 0,E6 0}
;ENDFOLD

;FOLD PLACE 6
DECL E6POS P1_23Smarties_6_App1={X 1022.18218,Y -949.33572,Z 1158.22,A 90,B 0,C -180,S 2,T 34,E1 0,E2 0,E3 0,E4 0,E5 0,E6 0}
DECL E6POS P1_23Smarties_6_App2={X 1022.18236,Y -949.33572,Z 958.217,A 90,B 0,C 180,S 2,T 34,E1 0,E2 0,E3 0,E4 0,E5 0,E6 0}
DECL E6POS P1_23Smarties_6_Place={X 972.18236,Y -999.33572,Z 858.218,A 90,B 0,C -180,S 2,T 34,E1 0,E2 0,E3 0,E4 0,E5 0,E6 0}
;ENDFOLD

;FOLD PLACE 7
DECL E6POS P1_23Smarties_7_App1={X 552.18218,Y -445.33572,Z 1158.22,A 90,B 0,C -180,S 2,T 2,E1 0,E2 0,E3 0,E4 0,E5 0,E6 0}
DECL E6POS P1_23Smarties_7_App2={X 552.18236,Y -445.33572,Z 958.217,A 90,B 0,C 180,S 2,T 2,E1 0,E2 0,E3 0,E4 0,E5 0,E6 0}
DECL E6POS P1_23Smarties_7_Place={X 502.18236,Y -495.33572,Z 858.218,A 90,B 0,C -180,S 2,T 2,E1 0,E2 0,E3 0,E4 0,E5 0,E6 0}
;ENDFOLD

;FOLD PLACE 8
DECL E6POS P1_23Smarties_8_App1={X 1022.18218,Y -445.33572,Z 1158.22,A 90,B 0,C -180,S 2,T 34,E1 0,E2 0,E3 0,E4 0,E5 0,E6 0}
DECL E6POS P1_23Smarties_8_App2={X 1022.18236,Y -445.33572,Z 958.217,A 90,B 0,C 180,S 2,T 34,E1 0,E2 0,E3 0,E4 0,E5 0,E6 0}
DECL E6POS P1_23Smarties_8_Place={X 972.18236,Y -495.33572,Z 858.218,A 90,B 0,C -180,S 2,T 34,E1 0,E2 0,E3 0,E4 0,E5 0,E6 0}
;ENDFOLD

;ENDFOLD

;FOLD Pallet 1 - Produto 22KitKat
;FOLD PLACE 1
DECL E6POS P1_22KitKat_1_App1={X 1066.23954,Y -442.43144,Z 1141.50207,A 180,B 0,C -180,S 2,T 2,E1 0,E2 0,E3 0,E4 0,E5 0,E6 0}
DECL E6POS P1_22KitKat_1_App2={X 1066.23956,Y -442.43156,Z 941.50237,A -180,B 0,C -180,S 2,T 2,E1 0,E2 0,E3 0,E4 0,E5 0,E6 0}
DECL E6POS P1_22KitKat_1_Place={X 1166.24033,Y -442.43147,Z 841.5026,A 180,B 0,C -180,S 2,T 2,E1 0,E2 0,E3 0,E4 0,E5 0,E6 0}
;ENDFOLD

;FOLD PLACE 2
DECL E6POS P1_22KitKat_2_App1={X 672.23958,Y -442.43157,Z 1141.50224,A -180,B 0,C -180,S 2,T 2,E1 0,E2 0,E3 0,E4 0,E5 0,E6 0}
DECL E6POS P1_22KitKat_2_App2={X 672.23959,Y -442.43151,Z 941.50181,A 180,B 0,C -180,S 2,T 2,E1 0,E2 0,E3 0,E4 0,E5 0,E6 0}
DECL E6POS P1_22KitKat_2_Place={X 772.24013,Y -442.43149,Z 841.50209,A -180,B 0,C 180,S 2,T 2,E1 0,E2 0,E3 0,E4 0,E5 0,E6 0}
;ENDFOLD

;FOLD PLACE 3
DECL E6POS P1_22KitKat_3_App1={X 328.23969,Y -442.43126,Z 1141.50239,A -180,B 0,C -180,S 2,T 2,E1 0,E2 0,E3 0,E4 0,E5 0,E6 0}
DECL E6POS P1_22KitKat_3_App2={X 328.23968,Y -442.4315,Z 941.50171,A -180,B 0,C -180,S 2,T 2,E1 0,E2 0,E3 0,E4 0,E5 0,E6 0}
DECL E6POS P1_22KitKat_3_Place={X 378.23966,Y -442.43116,Z 841.50213,A -180,B 0,C -180,S 2,T 2,E1 0,E2 0,E3 0,E4 0,E5 0,E6 0}
;ENDFOLD

;FOLD PLACE 4
DECL E6POS P1_22KitKat_4_App1={X 563.719,Y -340.46315,Z 1167.90223,A 90,B 0,C -180,S 2,T 2,E1 0,E2 0,E3 0,E4 0,E5 0,E6 0}
DECL E6POS P1_22KitKat_4_App2={X 563.71898,Y -340.46313,Z 1041.51054,A 90,B 0,C 180,S 2,T 2,E1 0,E2 0,E3 0,E4 0,E5 0,E6 0}
DECL E6POS P1_22KitKat_4_Place={X 563.71898,Y -390.46313,Z 841.51054,A 90,B 0,C 180,S 2,T 2,E1 0,E2 0,E3 0,E4 0,E5 0,E6 0}
;ENDFOLD

;FOLD PLACE 5
DECL E6POS P1_22KitKat_5_App1={X 563.71689,Y -818.63165,Z 1067.9,A 90,B 0,C 180,S 2,T 2,E1 0,E2 0,E3 0,E4 0,E5 0,E6 0}
DECL E6POS P1_22KitKat_5_App2={X 563.71689,Y -818.63117,Z 967.902,A 90,B 0,C 180,S 2,T 2,E1 0,E2 0,E3 0,E4 0,E5 0,E6 0}
DECL E6POS P1_22KitKat_5_Place={X 563.71689,Y -972.44848,Z 841.502,A 90,B 0,C 180,S 2,T 2,E1 0,E2 0,E3 0,E4 0,E5 0,E6 0}
;ENDFOLD

;FOLD PLACE 6
DECL E6POS P1_22KitKat_6_App1={X 1116.24408,Y -19.43165,Z 1117.9,A 180,B 0,C 180,S 2,T 2,E1 0,E2 0,E3 0,E4 0,E5 0,E6 0}
DECL E6POS P1_22KitKat_6_App2={X 1116.24382,Y -19.43206,Z 967.902,A -180,B 0,C 180,S 2,T 2,E1 0,E2 0,E3 0,E4 0,E5 0,E6 0}
DECL E6POS P1_22KitKat_6_Place={X 1166.24382,Y -69.43206,Z 841.503,A -180,B 0,C -180,S 2,T 2,E1 0,E2 0,E3 0,E4 0,E5 0,E6 0}
;ENDFOLD

;FOLD PLACE 7
DECL E6POS P1_22KitKat_7_App1={X 721.67971,Y -19.4321,Z 1117.9,A -180,B 0,C -180,S 2,T 2,E1 0,E2 0,E3 0,E4 0,E5 0,E6 0}
DECL E6POS P1_22KitKat_7_App2={X 721.67991,Y -19.43206,Z 967.902,A -180,B 0,C 180,S 2,T 2,E1 0,E2 0,E3 0,E4 0,E5 0,E6 0}
DECL E6POS P1_22KitKat_7_Place={X 771.67991,Y -69.43206,Z 841.5,A -180,B 0,C 180,S 2,T 2,E1 0,E2 0,E3 0,E4 0,E5 0,E6 0}
;ENDFOLD

;FOLD PLACE 8
DECL E6POS P1_22KitKat_8_App1={X 325.24357,Y -19.43175,Z 1117.9,A 180,B 0,C 180,S 2,T 2,E1 0,E2 0,E3 0,E4 0,E5 0,E6 0}
DECL E6POS P1_22KitKat_8_App2={X 325.2435,Y -19.43175,Z 967.902,A -180,B 0,C 180,S 2,T 2,E1 0,E2 0,E3 0,E4 0,E5 0,E6 0}
DECL E6POS P1_22KitKat_8_Place={X 375.2435,Y -69.43175,Z 841.502,A -180,B 0,C 180,S 2,T 2,E1 0,E2 0,E3 0,E4 0,E5 0,E6 0}
;ENDFOLD

;ENDFOLD

;FOLD Pallet 1 - Produto 24a28All
;FOLD PLACE 1
DECL E6POS P1_24a28All_1_App1={X 601.49375,Y -923.89214,Z 1014.54353,A 90,B 0,C 180,S 2,T 2,E1 0,E2 0,E3 0,E4 0,E5 0,E6 0}
DECL E6POS P1_24a28All_1_App2={X 601.49376,Y -923.89208,Z 914.54385,A 90,B 0,C 180,S 2,T 2,E1 0,E2 0,E3 0,E4 0,E5 0,E6 0}
DECL E6POS P1_24a28All_1_Place={X 601.49345,Y -1023.89188,Z 814.54423,A 90,B 0,C -180,S 2,T 2,E1 0,E2 0,E3 0,E4 0,E5 0,E6 0}
;ENDFOLD

;FOLD PLACE 2
DECL E6POS P1_24a28All_2_App1={X 601.49373,Y -618.89227,Z 1014.54432,A 90,B 0,C 180,S 2,T 2,E1 0,E2 0,E3 0,E4 0,E5 0,E6 0}
DECL E6POS P1_24a28All_2_App2={X 601.49376,Y -618.8921,Z 914.54396,A 90,B 0,C 180,S 2,T 2,E1 0,E2 0,E3 0,E4 0,E5 0,E6 0}
DECL E6POS P1_24a28All_2_Place={X 601.48326,Y -718.88641,Z 814.55074,A 90,B 0,C -180,S 2,T 2,E1 0,E2 0,E3 0,E4 0,E5 0,E6 0}
;ENDFOLD

;FOLD PLACE 3
DECL E6POS P1_24a28All_3_App1={X 601.49359,Y -313.892,Z 1014.54385,A 90,B 0,C -180,S 2,T 2,E1 0,E2 0,E3 0,E4 0,E5 0,E6 0}
DECL E6POS P1_24a28All_3_App2={X 601.49356,Y -313.89218,Z 914.54373,A 90,B 0,C 180,S 2,T 2,E1 0,E2 0,E3 0,E4 0,E5 0,E6 0}
DECL E6POS P1_24a28All_3_Place={X 601.49408,Y -413.89184,Z 814.54386,A 90,B 0,C -180,S 2,T 2,E1 0,E2 0,E3 0,E4 0,E5 0,E6 0}
;ENDFOLD

;ENDFOLD

;FOLD Pallet 1 - Produto 30All
;FOLD PLACE 1
DECL E6POS P1_30All_1_App1={X 1121.61951,Y -406.47558,Z 1014.58087,A -180,B 0,C 180,S 2,T 2,E1 0,E2 0,E3 0,E4 0,E5 0,E6 0}
DECL E6POS P1_30All_1_App2={X 1121.61952,Y -406.47565,Z 914.58052,A -180,B 0,C 180,S 2,T 2,E1 0,E2 0,E3 0,E4 0,E5 0,E6 0}
DECL E6POS P1_30All_1_Place={X 1221.62029,Y -406.47588,Z 814.58116,A -180,B 0,C 180,S 2,T 2,E1 0,E2 0,E3 0,E4 0,E5 0,E6 0}
;ENDFOLD

;FOLD PLACE 2
DECL E6POS P1_30All_2_App1={X 841.61889,Y -406.47587,Z 1014.58085,A -180,B 0,C 180,S 2,T 2,E1 0,E2 0,E3 0,E4 0,E5 0,E6 0}
DECL E6POS P1_30All_2_App2={X 841.61889,Y -406.47591,Z 914.5811,A -180,B 0,C 180,S 2,T 2,E1 0,E2 0,E3 0,E4 0,E5 0,E6 0}
DECL E6POS P1_30All_2_Place={X 941.61934,Y -406.47549,Z 814.58096,A -180,B 0,C 180,S 2,T 2,E1 0,E2 0,E3 0,E4 0,E5 0,E6 0}
;ENDFOLD

;FOLD PLACE 3
DECL E6POS P1_30All_3_App1={X 561.61985,Y -406.47561,Z 1014.58106,A -180,B 0,C 180,S 2,T 2,E1 0,E2 0,E3 0,E4 0,E5 0,E6 0}
DECL E6POS P1_30All_3_App2={X 561.61982,Y -406.47581,Z 914.58075,A -180,B 0,C -180,S 2,T 2,E1 0,E2 0,E3 0,E4 0,E5 0,E6 0}
DECL E6POS P1_30All_3_Place={X 661.61919,Y -406.47586,Z 814.58067,A -180,B 0,C 180,S 2,T 2,E1 0,E2 0,E3 0,E4 0,E5 0,E6 0}
;ENDFOLD

;FOLD PLACE 4
DECL E6POS P1_30All_4_App1={X 331.61953,Y -406.47631,Z 1014.58089,A 180,B 0,C 180,S 2,T 2,E1 0,E2 0,E3 0,E4 0,E5 0,E6 0}
DECL E6POS P1_30All_4_App2={X 331.61926,Y -406.47595,Z 914.58081,A -180,B 0,C 180,S 2,T 2,E1 0,E2 0,E3 0,E4 0,E5 0,E6 0}
DECL E6POS P1_30All_4_Place={X 381.61985,Y -406.47563,Z 814.58067,A -180,B 0,C 180,S 2,T 2,E1 0,E2 0,E3 0,E4 0,E5 0,E6 0}
;ENDFOLD

;ENDFOLD

;FOLD Pallet 1 - Produto 16CoffeCrisp
;FOLD PLACE 1
DECL E6POS P1_16CoffeCrisp_1_App1={X 1200.43974,Y -397.8314,Z 1019.00144,A -180,B 0,C -180,S 2,T 2,E1 0,E2 0,E3 0,E4 0,E5 0,E6 0}
DECL E6POS P1_16CoffeCrisp_1_App2={X 1200.43966,Y -397.83162,Z 892.60201,A -180,B 0,C -180,S 2,T 2,E1 0,E2 0,E3 0,E4 0,E5 0,E6 0}
DECL E6POS P1_16CoffeCrisp_1_Place={X 1262.09632,Y -407.70695,Z 814.59915,A 180,B 0,C -180,S 2,T 2,E1 0,E2 0,E3 0,E4 0,E5 0,E6 0}
;ENDFOLD

;FOLD PLACE 2
DECL E6POS P1_16CoffeCrisp_2_App1={X 799.43968,Y -397.83134,Z 1019.00144,A -180,B 0,C -180,S 2,T 2,E1 0,E2 0,E3 0,E4 0,E5 0,E6 0}
DECL E6POS P1_16CoffeCrisp_2_App2={X 799.43989,Y -397.8315,Z 892.60174,A -180,B 0,C -180,S 2,T 2,E1 0,E2 0,E3 0,E4 0,E5 0,E6 0}
DECL E6POS P1_16CoffeCrisp_2_Place={X 861.09619,Y -407.70679,Z 814.59921,A 180,B 0,C -180,S 2,T 2,E1 0,E2 0,E3 0,E4 0,E5 0,E6 0}
;ENDFOLD

;FOLD PLACE 3
DECL E6POS P1_16CoffeCrisp_3_App1={X 398.43885,Y -397.83136,Z 1019.00144,A 180,B 0,C -180,S 2,T 2,E1 0,E2 0,E3 0,E4 0,E5 0,E6 0}
DECL E6POS P1_16CoffeCrisp_3_App2={X 398.4393,Y -397.8311,Z 892.60169,A 180,B 0,C -180,S 2,T 2,E1 0,E2 0,E3 0,E4 0,E5 0,E6 0}
DECL E6POS P1_16CoffeCrisp_3_Place={X 460.09604,Y -407.70686,Z 814.59882,A -180,B 0,C -180,S 2,T 2,E1 0,E2 0,E3 0,E4 0,E5 0,E6 0}
;ENDFOLD

;FOLD PLACE 4
DECL E6POS P1_16CoffeCrisp_4_App1={X 603.92217,Y -417.5435,Z 1019.00139,A 90,B 0,C -180,S 2,T 2,E1 0,E2 0,E3 0,E4 0,E5 0,E6 0}
DECL E6POS P1_16CoffeCrisp_4_App2={X 603.92197,Y -417.54366,Z 969.00182,A 90,B 0,C -180,S 2,T 2,E1 0,E2 0,E3 0,E4 0,E5 0,E6 0}
DECL E6POS P1_16CoffeCrisp_4_Place={X 603.92197,Y -467.54366,Z 814.59924,A 90,B 0,C 180,S 2,T 2,E1 0,E2 0,E3 0,E4 0,E5 0,E6 0}
;ENDFOLD

;FOLD PLACE 5
DECL E6POS P1_16CoffeCrisp_5_App1={X 603.91816,Y -1017.52783,Z 1084.5782,A 90,B 0,C -180,S 2,T 2,E1 0,E2 0,E3 0,E4 0,E5 0,E6 0}
DECL E6POS P1_16CoffeCrisp_5_App2={X 603.91847,Y -1017.52787,Z 1064.57666,A 90,B 0,C -180,S 2,T 2,E1 0,E2 0,E3 0,E4 0,E5 0,E6 0}
DECL E6POS P1_16CoffeCrisp_5_Place={X 603.91847,Y -1067.52787,Z 964.58385,A 90,B 0,C -180,S 2,T 2,E1 0,E2 0,E3 0,E4 0,E5 0,E6 0}
;ENDFOLD

;FOLD PLACE 6
DECL E6POS P1_16CoffeCrisp_6_App1={X 1212.09935,Y 43.31562,Z 1014.58,A 180,B 0,C -180,S 2,T 2,E1 0,E2 0,E3 0,E4 0,E5 0,E6 0}
DECL E6POS P1_16CoffeCrisp_6_App2={X 1212.09951,Y 43.3156,Z 914.598,A -180,B 0,C -180,S 2,T 2,E1 0,E2 0,E3 0,E4 0,E5 0,E6 0}
DECL E6POS P1_16CoffeCrisp_6_Place={X 1262.09953,Y -6.68448,Z 814.597,A -180,B 0,C -180,S 2,T 2,E1 0,E2 0,E3 0,E4 0,E5 0,E6 0}
;ENDFOLD

;FOLD PLACE 7
DECL E6POS P1_16CoffeCrisp_7_App1={X 811.09401,Y 43.32527,Z 1014.58,A 180,B 0,C -180,S 2,T 2,E1 0,E2 0,E3 0,E4 0,E5 0,E6 0}
DECL E6POS P1_16CoffeCrisp_7_App2={X 811.09421,Y 43.32547,Z 914.598,A -180,B 0,C -180,S 2,T 2,E1 0,E2 0,E3 0,E4 0,E5 0,E6 0}
DECL E6POS P1_16CoffeCrisp_7_Place={X 861.09421,Y -6.67453,Z 814.605,A 180,B 0,C -180,S 2,T 2,E1 0,E2 0,E3 0,E4 0,E5 0,E6 0}
;ENDFOLD

;FOLD PLACE 8
DECL E6POS P1_16CoffeCrisp_8_App1={X 410.09442,Y 43.3219,Z 1014.6,A -180,B 0,C -180,S 2,T 2,E1 0,E2 0,E3 0,E4 0,E5 0,E6 0}
DECL E6POS P1_16CoffeCrisp_8_App2={X 410.09442,Y 43.32219,Z 914.6,A 180,B 0,C -180,S 2,T 2,E1 0,E2 0,E3 0,E4 0,E5 0,E6 0}
DECL E6POS P1_16CoffeCrisp_8_Place={X 460.09442,Y -6.67781,Z 814.608,A -180,B 0,C -180,S 2,T 2,E1 0,E2 0,E3 0,E4 0,E5 0,E6 0}
;ENDFOLD

;ENDFOLD

;FOLD Pallet 1 - Produto 10CoffeCrisp
;FOLD PLACE 1
DECL E6POS P1_10CoffeCrisp_1_App1={X 678.21322,Y -939.58995,Z 1064.60195,A 90,B 0,C -180,S 2,T 2,E1 0,E2 0,E3 0,E4 0,E5 0,E6 0}
DECL E6POS P1_10CoffeCrisp_1_App2={X 678.21325,Y -939.58998,Z 964.60203,A 90,B 0,C -180,S 2,T 2,E1 0,E2 0,E3 0,E4 0,E5 0,E6 0}
DECL E6POS P1_10CoffeCrisp_1_Place={X 678.21325,Y -1039.58982,Z 814.60187,A 90,B 0,C -180,S 2,T 2,E1 0,E2 0,E3 0,E4 0,E5 0,E6 0}
;ENDFOLD

;FOLD PLACE 2
DECL E6POS P1_10CoffeCrisp_2_App1={X 678.21396,Y -459.58981,Z 1064.60195,A 90,B 0,C -180,S 2,T 2,E1 0,E2 0,E3 0,E4 0,E5 0,E6 0}
DECL E6POS P1_10CoffeCrisp_2_App2={X 678.21406,Y -459.59,Z 964.60191,A 90,B 0,C -180,S 2,T 2,E1 0,E2 0,E3 0,E4 0,E5 0,E6 0}
DECL E6POS P1_10CoffeCrisp_2_Place={X 678.21406,Y -559.59017,Z 814.6021,A 90,B 0,C -180,S 2,T 2,E1 0,E2 0,E3 0,E4 0,E5 0,E6 0}
;ENDFOLD

